# B&R Automation Studio project NAELD004C00R10L518F00 (part 24)

#### Act_Link.st
```iecst
(** 2019-01-07 **)
ACTION Act_Link:

	IF EDGEPOS(p_tyLinkUSSMEMA1AlmData.udiCode <> 0) THEN
		p_tyLinkUSSMEMA1AlmData.sProgNm	:= 'Mag1_1';
		p_tyLinkUSSMEMA1AlmData.sAlmMsg	:= 'Pulling Board Failed';
	END_IF

	IF EDGEPOS(p_tyLinkUSSMEMA2AlmData.udiCode <> 0) THEN
		p_tyLinkUSSMEMA2AlmData.sProgNm	:= 'Mag2_1';
		p_tyLinkUSSMEMA2AlmData.sAlmMsg	:= 'Pulling Board Failed';
	END_IF

	IF EDGEPOS(p_tyLinkUSSMEMA3AlmData.udiCode <> 0) THEN
		p_tyLinkUSSMEMA3AlmData.sProgNm	:= 'Mag3_1';
		p_tyLinkUSSMEMA3AlmData.sAlmMsg	:= 'Pulling Board Failed';
	END_IF

	IF EDGEPOS(p_tyLinkDSSMEMA1AlmData.udiCode <> 0) THEN
		p_tyLinkDSSMEMA1AlmData.sProgNm	:= 'Mag1_2';
		p_tyLinkDSSMEMA1AlmData.sAlmMsg	:= 'Pulling Board Failed';
	END_IF

	IF EDGEPOS(p_tyLinkDSSMEMA2AlmData.udiCode <> 0) THEN
		p_tyLinkDSSMEMA2AlmData.sProgNm	:= 'Mag2_2';
		p_tyLinkDSSMEMA2AlmData.sAlmMsg	:= 'Pulling Board Failed';
	END_IF

	IF EDGEPOS(p_tyLinkDSSMEMA3AlmData.udiCode <> 0) THEN
		p_tyLinkDSSMEMA3AlmData.sProgNm	:= 'Mag3_2';
		p_tyLinkDSSMEMA3AlmData.sAlmMsg	:= 'Pulling Board Failed';
	END_IF

	//Index 1 For Internal Use

	pa_tyAlmData[2]		:= p_tyLinkUsrFolderAlmData;
	pa_tyAlmData[3]		:= p_tyLinkLibVerAlmData;
	pa_tyAlmData[4]		:= p_tyLinkTimeAlmData;
	pa_tyAlmData[5]		:= p_tyLinkTimeAlmData1;
	pa_tyAlmData[6]		:= p_tyLinkHWInfoAlmData;
	pa_tyAlmData[7]		:= p_tyLinkProdRcpAlmData;
	pa_tyAlmData[8]		:= p_tyLinkMpProdRcpAlmData;
	pa_tyAlmData[9]		:= p_tyLinkMagRcpAlmData;
	pa_tyAlmData[10]	:= p_tyLinkMagRcpAlmData1;

	pa_tyAlmData[11]	:= p_tyLinkMcParamAlmData;
	pa_tyAlmData[12]	:= p_tyLinkNtParamAlmData;
	pa_tyAlmData[13]	:= p_tyLinkUsrMgmtAlmData;
	pa_tyAlmData[14]	:= p_tyLinkBuffer1AlmData;
	pa_tyAlmData[15]	:= p_tyLinkBuffer2AlmData;
	pa_tyAlmData[16]	:= p_tyLinkBuffer3AlmData;
	pa_tyAlmData[17]	:= p_tyLinkBuffer4AlmData;
	pa_tyAlmData[18]	:= p_tyLinkUSSMEMA1AlmData;
	pa_tyAlmData[19]	:= p_tyLinkUSSMEMA2AlmData;
	pa_tyAlmData[20]	:= p_tyLinkUSSMEMA3AlmData;
	pa_tyAlmData[21]	:= p_tyLinkUSSMEMA4AlmData;
	pa_tyAlmData[22]	:= p_tyLinkDSSMEMA1AlmData;
	pa_tyAlmData[23]	:= p_tyLinkDSSMEMA2AlmData;
	pa_tyAlmData[24]	:= p_tyLinkDSSMEMA3AlmData;
	pa_tyAlmData[25]	:= p_tyLinkDSSMEMA4AlmData;

	pa_tyAlmData[26]	:= p_tyLinkDSSMEMAAAlmData;
	pa_tyAlmData[27]	:= p_tyLinkDSSMEMABAlmData;
	pa_tyAlmData[28]	:= p_tyLinkInShutterAlmData;
	pa_tyAlmData[29]	:= p_tyLinkOutShutterAlmData;
	pa_tyAlmData[30]	:= p_tyLinkPullerAlmData;
	pa_tyAlmData[31]	:= p_tyLinkPullConvAlmData;
	pa_tyAlmData[32]	:= p_tyLinkMagConv1AlmData;
	pa_tyAlmData[33]	:= p_tyLinkMagConv2AlmData;
	pa_tyAlmData[34]	:= p_tyLinkMagConv3AlmData;
	pa_tyAlmData[35]	:= p_tyLinkMagConv4AlmData;

	pa_tyAlmData[36]	:= p_tyLinkAWOpenAlmData;
	pa_tyAlmData[37]	:= p_tyLinkAWOpenAlmData1;
	pa_tyAlmData[38]	:= p_tyLinkAWOpenAlmData2;
	pa_tyAlmData[39]	:= p_tyLinkAWOpenAlmData3;
	pa_tyAlmData[40]	:= p_tyLinkTravAlmData;
	pa_tyAlmData[41]	:= p_tyLinkTravAlmData1;
	pa_tyAlmData[42]	:= p_tyLinkTravAlmData2;
	pa_tyAlmData[43]	:= p_tyLinkTravAlmData3;
	pa_tyAlmData[44]	:= p_tyLinkLifterBtmAlmData;
	pa_tyAlmData[45]	:= p_tyLinkLifterBtmAlmData1;
	pa_tyAlmData[46]	:= p_tyLinkLifterBtmAlmData2;
	pa_tyAlmData[47]	:= p_tyLinkLifterBtmAlmData3;
	pa_tyAlmData[48]	:= p_tyLinkDIAlmData1;
	pa_tyAlmData[49]	:= p_tyLinkDIAlmData2;
	pa_tyAlmData[50]	:= p_tyLinkDIAlmData3;
	pa_tyAlmData[51]	:= p_tyLinkDIAlmData4;

	pa_tyAlmData[52]	:= p_tyLinkAGVMag1AlmData;
	pa_tyAlmData[53]	:= p_tyLinkAGVMag2AlmData;
	pa_tyAlmData[54]	:= p_tyLinkAGVMag3AlmData;
	pa_tyAlmData[55]	:= p_tyLinkAGVMag4AlmData;

	pa_tyAlmData[56]	:= p_tyLinkHermesAlmData;
	pa_tyAlmData[57]	:= p_tyLinkDSHermesAAlmData;
	pa_tyAlmData[58]	:= p_tyLinkDSHermesAAlmData1;
	pa_tyAlmData[59]	:= p_tyLinkDSHermesAAlmData2;
	pa_tyAlmData[60]	:= p_tyLinkDSHermesAAlmData3;
	pa_tyAlmData[61]	:= p_tyLinkDSHermesAAlmData4;

	pa_tyAlmData[62]	:= p_tyLinkDSHermesBAlmData;
	pa_tyAlmData[63]	:= p_tyLinkDSHermesBAlmData1;
	pa_tyAlmData[64]	:= p_tyLinkDSHermesBAlmData2;
	pa_tyAlmData[65]	:= p_tyLinkDSHermesBAlmData3;
	pa_tyAlmData[66]	:= p_tyLinkDSHermesBAlmData4;

	pa_tyAlmData[67]	:= p_tyLinkRmtHermesAlmData;
	pa_tyAlmData[68]	:= p_tyLinkRmtHermesAlmData1;
	pa_tyAlmData[69]	:= p_tyLinkRmtHermesAlmData2;
	pa_tyAlmData[70]	:= p_tyLinkRmtHermesAlmData3;
	pa_tyAlmData[71]	:= p_tyLinkLFLeaderAlmData;
	pa_tyAlmData[72]	:= p_tyLinkLFFollowerAlmData;
	pa_tyAlmData[73]	:= p_tyLinkLFFollowerInfoData;
	pa_tyAlmData[74]	:= p_tyLinkLFFollowerInfoData1;
	pa_tyAlmData[75]	:= p_tyLinkFollower1AlmData;
	pa_tyAlmData[76]	:= p_tyLinkFollower1InfoData;
	pa_tyAlmData[77]	:= p_tyLinkFollower1InfoData1;
	pa_tyAlmData[78]	:= p_tyLinkFollower2AlmData;
	pa_tyAlmData[79]	:= p_tyLinkFollower2InfoData;
	pa_tyAlmData[80]	:= p_tyLinkFollower2InfoData1;
	pa_tyAlmData[81]	:= p_tyLinkLCSMngRcpAlmData;
	pa_tyAlmData[82]	:= p_tyLinkLCSLFAlmData;
	pa_tyAlmData[83]	:= p_tyLinkLCSLFInfoData;
	pa_tyAlmData[84]	:= p_tyLinkOpsTravLifLDAlmData;

	pa_tyAlmData[85]	:= p_tyLinkPPAlmData;
	pa_tyAlmData[86]	:= p_tyLinkPPAlmData1;
	pa_tyAlmData[87]	:= p_tyLinkPPAlmData2;
	pa_tyAlmData[89]	:= p_tyLinkPPAlmData3;
//	pa_tyAlmData[90]	:= p_tyLinkOpsMagLD3AlmData;
//	pa_tyAlmData[91]	:= p_tyLinkOpsMagLD3AlmData1;
//	pa_tyAlmData[92]	:= p_tyLinkOpsMagLD4AlmData;
//	pa_tyAlmData[93]	:= p_tyLinkOpsMagLD4AlmData1;
	pa_tyAlmData[94]	:= p_tyLinkOpsLifMagLDAlmData;
	pa_tyAlmData[95]	:= p_tyLinkOpsLifMagLDAlmData1;

	pa_tyAlmData[96]	:= p_tyLinkOpsMagConvLD1AlmData;
	pa_tyAlmData[97]	:= p_tyLinkOpsMagConvLD1AlmData1;
	pa_tyAlmData[98]	:= p_tyLinkOpsMagConvLD2AlmData;
	pa_tyAlmData[99]	:= p_tyLinkOpsMagConvLD2AlmData1;
	pa_tyAlmData[100]	:= p_tyLinkOpsMagConvLD3AlmData;
	pa_tyAlmData[101]	:= p_tyLinkOpsMagConvLD3AlmData1;
	pa_tyAlmData[102]	:= p_tyLinkOpsMagConvLD4AlmData;
	pa_tyAlmData[103]	:= p_tyLinkOpsMagConvLD4AlmData1;

	pa_tyAlmData[104]	:= p_tyLinkSelClamp1AlmData;
	pa_tyAlmData[105]	:= p_tyLinkSelClamp2AlmData;
	pa_tyAlmData[106]	:= p_tyLinkSelClamp3AlmData;
	pa_tyAlmData[107]	:= p_tyLinkSelClamp4AlmData;

	pa_tyAlmData[108]	:= p_tyLinkUSSOT1AlmData;
	pa_tyAlmData[109]	:= p_tyLinkUSSOT2AlmData;
	pa_tyAlmData[110]	:= p_tyLinkUSSOT3AlmData;
	pa_tyAlmData[111]	:= p_tyLinkUSSOT4AlmData;
	pa_tyAlmData[112]	:= p_tyLinkDSSOT1AlmData;
	pa_tyAlmData[113]	:= p_tyLinkDSSOT2AlmData;
	pa_tyAlmData[114]	:= p_tyLinkDSSOT3AlmData;
	pa_tyAlmData[115]	:= p_tyLinkDSSOT4AlmData;

	pa_tyAlmData[116]	:= p_tyLinkMcAlarmData;
	pa_tyAlmData[117]	:= p_tyLinkMc1AlarmData;

	pa_tyAlmData[118]	:= p_tyLinkUSBBarcodeAlmData;
	pa_tyAlmData[119]	:= p_tyLinkUSBBarcodeAlmData1;
	pa_tyAlmData[120]	:= p_tyLinkUSBBarcodeAlmData2;

	pa_tyAlmData[121]	:= p_tyLinkAGVAlmData1;
	pa_tyAlmData[122]	:= p_tyLinkRS232FrmAlmData;

	pa_tyAlmData[123]	:= p_tyLinkAWPushOrPullerAlmData;
	pa_tyAlmData[124]	:= p_tyLinkAWPushOrPullerAlmData1;
	pa_tyAlmData[125]	:= p_tyLinkAWPushOrPullerAlmData2;
	pa_tyAlmData[126]	:= p_tyLinkAWPushOrPullerAlmData3;
	pa_tyAlmData[127]	:= p_tyLinkMtrPshrAlmData;

	pa_tyAlmData[128]	:= p_tyLinkInShutterAlmData2;
	pa_tyAlmData[129]	:= p_tyLinkInShutterAlmData3;

	pa_tyAlmData[130]	:= p_tyLinkDIAlmData5;
	pa_tyAlmData[131]	:= p_tyLinkDIAlmData6;		//JOHN

//	pa_tyAlmData[131]	:= p_tyLinkUSHermesInfoData1;//new for Hermes 1.3
//	pa_tyAlmData[132]	:= p_tyLinkUSHermesInfoData2;//new for Hermes 1.3
//	pa_tyAlmData[133]	:= p_tyLinkUSHermesAlmData5;//new for Hermes 1.3
	pa_tyAlmData[134]	:= p_tyLinkRmtHermesInfoData;//new for Hermes 1.3
	pa_tyAlmData[135]	:= p_tyLinkSvyHermesAlmData;//new for Hermes 1.3
	pa_tyAlmData[136]	:= p_tyLinkSvyHermesAlmData1;//new for Hermes 1.3
	pa_tyAlmData[137]	:= p_tyLinkSvyHermesAlmData2;//new for Hermes 1.3
	pa_tyAlmData[138]	:= p_tyLinkSvyHermesAlmData3;//new for Hermes 1.3
	pa_tyAlmData[139]	:= p_tyLinkSvyHermesInfoData;//new for Hermes 1.3
	pa_tyAlmData[140]	:= p_tyLinkSvyHermesInfoData1;//new for Hermes 1.3
	pa_tyAlmData[141]	:= p_tyLinkSvyHermesInfoData2;//new for Hermes 1.3
	pa_tyAlmData[142]	:= p_tyLinkSvyHermesInfoData3;//new for Hermes 1.3
	pa_tyAlmData[143]	:= p_tyLinkSvyHermesAlmData4;//new for Hermes 1.3
	pa_tyAlmData[144]	:= p_tyLinkSvyHermesInfoData4;//new for Hermes 1.3

	pa_tyAlmData[145]	:= p_tyLinkAutoRcpAlmData;
	pa_tyAlmData[146]	:= p_tyLinkAutoRcpInfoData;
	pa_tyAlmData[147]	:= p_tyLinkAutoRcpInfoData1;
	pa_tyAlmData[148]	:= p_tyLinkOutShutterAlmData2;
	pa_tyAlmData[149]	:= p_tyLinkTrllyAlmData;
	pa_tyAlmData[150]	:= p_tyLinkTrlly2AlmData;

END_ACTION
```

#### Act_LinkAction.st
```iecst
(** 2019-03-29 **)
ACTION Act_LinkAction:

	//Delete Old Log File for 24 hours After Machine is Continuous Running 30 Days.

	fbDlyTmr(IN := TRUE);
	IF fbDlyTmr.Q THEN
		fbDeleteLogTmr (IN := TRUE);
		IF fbDeleteLogTmr.Q AND eStatus <> Busy THEN
			p_eAct := AlarmActDeleteOldLog;
			IF eStat = AlarmActDeleteOldLog AND eStatus = Done THEN
				p_eAct := AlarmActIdle;
				fbDlyTmr (IN := FALSE);
				fbDeleteLogTmr (IN := FALSE);
			END_IF
		END_IF
	END_IF

END_ACTION
```

#### Act_Main.st
```iecst
(** 2019-02-23 **)
ACTION Act_Main:

	//Main
	CASE eStat OF

		AlarmActIdle:
			IF eStatus <> Idle THEN	//Reset Data
				//Private
				fbDirCreate1(bEn := FALSE);
				fbDirCreate2(bEn := FALSE);
				fbFileOldDel1(bEn := FALSE);
				fbFileRead1(bEn := FALSE);
				fbFileAppend1(bEn := FALSE);
				fbFileWrite1(bEn := FALSE);
				usiStep	:= 0;

				bHistoryFileNotFound	:= FALSE;
				udiWriteLogCntr			:= 1;

				sStatTxt	:= a_sStatText[eStat];

			END_IF

			eStatus	:= Idle;

		AlarmActCreateDir:
			IF eStatus = Idle OR eStatus = Busy THEN

				eStatus	:= Busy;

				sStatTxt	:= a_sStatText[eStat];

				CASE usiStep OF
					0:
						fbDirCreate1(bEn := TRUE);
						IF fbDirCreate1.udiStatus = 0 THEN
							usiStep	:= 1;
						ELSIF fbDirCreate1.udiStatus < 65534 THEN
							eStatus		:= Error;

							IF fbDirCreate1.udiStatus = 1908 THEN
								udiStatus	:= 10000;	//Create User Directory Error
							ELSE
								udiStatus	:= fbDirCreate1.udiStatus;
							END_IF
						END_IF

					1:
						fbDirCreate2(bEn := TRUE);
						IF fbDirCreate2.udiStatus = 0 THEN
							eStatus	:= Done;
						ELSIF fbDirCreate2.udiStatus < 65534 THEN
							eStatus		:= Error;

							IF fbDirCreate2.udiStatus = 1908 THEN
								udiStatus	:= 10001;	//Create Alarm Directory Error
							ELSE
								udiStatus	:= fbDirCreate2.udiStatus;
							END_IF
						END_IF

				END_CASE

			END_IF

		AlarmActDeleteOldLog:
			IF eStatus = Idle OR eStatus = Busy THEN

				eStatus	:= Busy;

				sStatTxt	:= a_sStatText[eStat];

				fbFileOldDel1.dtDTNow			:= p_dtCurrDT;
				fbFileOldDel1.udiFileKeepDay	:= p_udiFileKeepDay;
				fbFileOldDel1(bEn := TRUE);
				IF fbFileOldDel1.udiStatus = 0 THEN
					eStatus	:= Done;
				ELSIF fbFileOldDel1.udiStatus < 65534 THEN
					eStatus		:= Error;

					IF fbFileOldDel1.udiStatus = 1910 THEN
						udiStatus	:= 10002;	//Get Directory Info Error While Deleting Old Log
					ELSIF fbFileOldDel1.udiStatus = 1911 THEN
						udiStatus	:= 10003;	//Directory Read Error While Deleting Old Log
					ELSIF fbFileOldDel1.udiStatus = 1912 THEN
						udiStatus	:= 10004;	//File Delete Error While Deleting Old Log
					ELSE
						udiStatus	:= fbFileOldDel1.udiStatus;
					END_IF
				END_IF

			END_IF

		AlarmActReadHistory:
			IF eStatus = Idle OR eStatus = Busy THEN

				eStatus	:= Busy;

				sStatTxt	:= a_sStatText[eStat];

				fbFileRead1(bEn := TRUE);
				IF fbFileRead1.udiStatus = 0 THEN
					eStatus	:= Done;
				ELSIF fbFileRead1.udiStatus < 65534 THEN
					eStatus		:= Error;

					IF fbFileRead1.udiStatus = 1900 THEN
						udiStatus	:= 10005;	//File Open Error While Reading Alarm History
					ELSIF fbFileRead1.udiStatus = 1902 THEN
						udiStatus	:= 10006;	//File Read Error While Reading Alarm History
					ELSIF fbFileRead1.udiStatus = 1904 THEN
						udiStatus	:= 10007;	//File Close Error While Reading Alarm History
					ELSIF fbFileRead1.udiStatus = 1915 THEN
						eStatus					:= Done;
						bHistoryFileNotFound	:= TRUE;
					ELSE
						udiStatus	:= fbFileRead1.udiStatus;
					END_IF
				END_IF

			END_IF

		AlarmActWriteHistory:
			IF eStatus = Idle OR eStatus = Busy THEN

				eStatus	:= Busy;

				sStatTxt	:= a_sStatText[eStat];

				fbFileWrite1(bEn := TRUE);
				IF fbFileWrite1.udiStatus = 0 THEN
					eStatus	:= Done;
				ELSIF fbFileWrite1.udiStatus < 65534 THEN
					eStatus		:= Error;

					IF fbFileWrite1.udiStatus = 1900 THEN
						udiStatus	:= 10008;	//File Open Error While Writing Alarm History
					ELSIF fbFileWrite1.udiStatus = 1901 THEN
						udiStatus	:= 10009;	//File Create Error While Writing Alarm History
					ELSIF fbFileWrite1.udiStatus = 1903 THEN
						udiStatus	:= 10010;	//File Write Error While Writing Alarm History
					ELSIF fbFileWrite1.udiStatus = 1904 THEN
						udiStatus	:= 10011;	//File Close Error While Writing Alarm History
					ELSIF fbFileWrite1.udiStatus = 1914 THEN
						udiStatus	:= 10012;	//Directory Does Not Exist While Writing Alarm History
					ELSE
						udiStatus	:= fbFileWrite1.udiStatus;
					END_IF
				END_IF

			END_IF

		AlarmActAppendLog:
			IF eStatus = Idle OR eStatus = Busy THEN

				eStatus	:= Busy;

				sStatTxt	:= a_sStatText[eStat];

				dtCurrDTTemp			:= p_dtCurrDT;
				fbFileAppend1.sFile		:= DT_TO_STRING(dtCurrDTTemp);
				fbFileAppend1.sFile		:= MID(fbFileAppend1.sFile , 10 , 4);
				fbFileAppend1.sFile		:= CONCAT('ALARM_' , fbFileAppend1.sFile);
				fbFileAppend1.sFile		:= CONCAT(fbFileAppend1.sFile , '.dat');

				fbFileAppend1.p_Src		:= ADR(a_sLogList[udiWriteLogCntr]);
				fbFileAppend1.udiLen	:= LEN(a_sLogList[udiWriteLogCntr]);

				fbFileAppend1(bEn := TRUE);
				IF fbFileAppend1.udiStatus = 0 THEN
					IF udiWriteLogCntr >= udiLogCntr THEN
						eStatus	:= Done;
					ELSE
						udiWriteLogCntr	:= udiWriteLogCntr + 1;
						fbFileAppend1(bEn := FALSE);
					END_IF

				ELSIF fbFileAppend1.udiStatus < 65534 THEN
					eStatus		:= Error;

					IF fbFileAppend1.udiStatus = 1900 THEN
						udiStatus	:= 10013;	//File Open Error While Writing Alarm Log
					ELSIF fbFileAppend1.udiStatus = 1901 THEN
						udiStatus	:= 10014;	//File Create Error While Writing Alarm Log
					ELSIF fbFileAppend1.udiStatus = 1913 THEN
						udiStatus	:= 10015;	//Get File Info Error While Writing Alarm Log
					ELSIF fbFileAppend1.udiStatus = 1903 THEN
						udiStatus	:= 10016;	//File Write Error While Writing Alarm Log
					ELSIF fbFileAppend1.udiStatus = 1904 THEN
						udiStatus	:= 10017;	//File Close Error While Writing Alarm Log
					ELSIF fbFileAppend1.udiStatus = 1914 THEN
						udiStatus	:= 10018;	//Directory Does Not Exist While Writing Alarm Log
					ELSE
						udiStatus	:= fbFileAppend1.udiStatus;
					END_IF
				END_IF

			END_IF

		AlarmActAppendLogWriteHistory:
			IF eStatus = Idle OR eStatus = Busy THEN

				eStatus	:= Busy;

				sStatTxt	:= a_sStatText[eStat];

				dtCurrDTTemp			:= p_dtCurrDT;
				fbFileAppend1.sFile		:= DT_TO_STRING(dtCurrDTTemp);
				fbFileAppend1.sFile		:= MID(fbFileAppend1.sFile , 10 , 4);
				fbFileAppend1.sFile		:= CONCAT('ALARM_' , fbFileAppend1.sFile);
				fbFileAppend1.sFile		:= CONCAT(fbFileAppend1.sFile , '.dat');

				fbFileAppend1.p_Src		:= ADR(a_sLogList[udiWriteLogCntr]);
				fbFileAppend1.udiLen	:= LEN(a_sLogList[udiWriteLogCntr]);

				fbFileAppend1(bEn := TRUE);
				fbFileWrite1(bEn := TRUE);

				IF (fbFileAppend1.udiStatus = 0) AND (udiWriteLogCntr >= udiLogCntr) AND fbFileWrite1.udiStatus = 0 THEN
					eStatus	:= Done;

				ELSIF fbFileAppend1.udiStatus = 0 AND udiWriteLogCntr < udiLogCntr THEN
					udiWriteLogCntr	:= udiWriteLogCntr + 1;
					fbFileAppend1(bEn := FALSE);

				ELSIF fbFileWrite1.udiStatus > 0 AND fbFileWrite1.udiStatus < 65534 THEN
					eStatus		:= Error;

					IF fbFileWrite1.udiStatus = 1900 THEN
						udiStatus	:= 10019;	//File Open Error While Writing Alarm History
					ELSIF fbFileWrite1.udiStatus = 1901 THEN
						udiStatus	:= 10020;	//File Create Error While Writing Alarm History
					ELSIF fbFileWrite1.udiStatus = 1903 THEN
						udiStatus	:= 10021;	//File Write Error While Writing Alarm History
					ELSIF fbFileWrite1.udiStatus = 1904 THEN
						udiStatus	:= 10022;	//File Close Error While Writing Alarm History
					ELSIF fbFileWrite1.udiStatus = 1914 THEN
						udiStatus	:= 10023;	//Directory Does Not Exist While Writing Alarm History
					ELSE
						udiStatus	:= fbFileWrite1.udiStatus;
					END_IF

				ELSIF fbFileAppend1.udiStatus > 0 AND fbFileAppend1.udiStatus < 65534 THEN
					eStatus		:= Error;

					IF fbFileAppend1.udiStatus = 1900 THEN
						udiStatus	:= 10024;	//File Open Error While Writing Alarm Log
					ELSIF fbFileAppend1.udiStatus = 1901 THEN
						udiStatus	:= 10025;	//File Create Error While Writing Alarm Log
					ELSIF fbFileAppend1.udiStatus = 1913 THEN
						udiStatus	:= 10026;	//Get File Info Error While Writing Alarm Log
					ELSIF fbFileAppend1.udiStatus = 1903 THEN
						udiStatus	:= 10027;	//File Write Error While Writing Alarm Log
					ELSIF fbFileAppend1.udiStatus = 1904 THEN
						udiStatus	:= 10028;	//File Close Error While Writing Alarm Log
					ELSIF fbFileAppend1.udiStatus = 1914 THEN
						udiStatus	:= 10029;	//Directory Does Not Exist While Writing Alarm Log
					ELSE
						udiStatus	:= fbFileAppend1.udiStatus;
					END_IF
				END_IF

			END_IF

		AlarmActResetHistory:
			IF eStatus = Idle OR eStatus = Busy THEN

				eStatus	:= Busy;

				sStatTxt	:= a_sStatText[eStat];

				memset(ADR(a_sHistoryList) , 0 , SIZEOF(a_sHistoryList));

				fbFileWrite1(bEn := TRUE);
				IF fbFileWrite1.udiStatus = 0 THEN
					eStatus	:= Done;
				ELSIF fbFileWrite1.udiStatus < 65534 THEN
					eStatus		:= Error;

					IF fbFileWrite1.udiStatus = 1900 THEN
						udiStatus	:= 10030;	//File Open Error While Resetting Alarm History
					ELSIF fbFileWrite1.udiStatus = 1901 THEN
						udiStatus	:= 10031;	//File Create Error While Resetting Alarm History
					ELSIF fbFileWrite1.udiStatus = 1903 THEN
						udiStatus	:= 10032;	//File Write Error While Resetting Alarm History
					ELSIF fbFileWrite1.udiStatus = 1904 THEN
						udiStatus	:= 10033;	//File Close Error While Resetting Alarm History
					ELSIF fbFileWrite1.udiStatus = 1914 THEN
						udiStatus	:= 10034;	//Directory Does Not Exist While Resetting Alarm History
					ELSE
						udiStatus	:= fbFileWrite1.udiStatus;
					END_IF
				END_IF

			END_IF

		AlarmActBGStartLog:
			IF eStatus = Idle OR eStatus = Busy THEN

				sStatTxt	:= a_sStatText[eStat];

				bAlarmLog	:= TRUE;
				eStatus		:= Done;

			END_IF

		AlarmActBGStopLog:
			IF eStatus = Idle OR eStatus = Busy THEN

				sStatTxt	:= a_sStatText[eStat];

				bAlarmLog	:= FALSE;
				eStatus		:= Done;

			END_IF

	END_CASE

END_ACTION
```

#### Act_RstErr.st
```iecst
(** 2020-07-27 **)
ACTION Act_RstErr:

	IF p_udiRstErr <> udiRstErrOld THEN
		bRstErr			:= TRUE;
		udiRstErrOld	:= p_udiRstErr;
	ELSE
		bRstErr			:= FALSE;
	END_IF

	//Checking which Warning is clear
	IF a_tyWarningCurrList[1].sMsg <> '' AND p_tyLinkLibVerAlmData.udiCode = 0 THEN

		FOR udi2 := 1 TO (udiWarningMax) DO
			udiRecorded1:= udiRecorded[udi2];
			IF 	(pa_tyAlmData[udiRecorded1].eSeverity =  AlmSeverityNA) AND udiRecorded1<> 0 THEN
				bRstWarning := TRUE;
				EXIT;
			ELSE
				bRstWarning := FALSE;
			END_IF

		END_FOR
	ELSE
		bRstWarning := FALSE;
	END_IF

END_ACTION
```

### ProdRcp.typ
```iecst
(*2020-07-24*)
(**)
(*Action*)

TYPE
	eProdRcpAction :
		(
		ProdRcpActIdle,
		ProdRcpActCreateDir,
		ProdRcpActAddEdit,
		ProdRcpActDel,
		ProdRcpActGetInfo,
		ProdRcpActGetList,
		ProdRcpActFilter,
		ProdRcpActLoadRcp,
		ProdRcpActAdd,
		ProdRcpActEdit,
		ProdRcpActReadCurrRcp,
		ProdRcpActWriteCurrRcpParam,
		ProdRcpActSaveList,
		ProdRcpActSort,
		ProdRcpActEndCharFilter
		);
END_TYPE

(**)
(*Data*)

TYPE
	tyProdRcpParam : 	STRUCT
		sRcpNm : STRING[254];
		diWidthInUM : DINT;
		diWidthInUM2 : DINT;
		diIntvlCntr : DINT;
		diMinSltValue : DINT;
		diMaxSltValue : DINT;
		diPitch : DINT;
		usiMcMod : USINT;
		usiFlippedBrd : USINT;
		bTopToBtm : BOOL;
		bLongBrd : BOOL;
		sDisplayInfo : STRING[30];
		dtLastModified : DATE_AND_TIME;
		diWidthInUMRear : DINT;
		diPitchRear : DINT;
		diMinSltValueRear : DINT;
		diMaxSltValueRear : DINT;
		diMtrPshrExtSpd : DINT; (*Puller*)
		diMtrPshrExtTorq : DINT;
		diPshrOffset : DINT;
	END_STRUCT;
END_TYPE
```

### ProdRcp.var
```iecst
(*2020-06-08*)
(**)
(*Constant*)
VAR CONSTANT
	c_udiProdRcpMax : UDINT := 2000;
END_VAR
(**)
(*Action & State & Status*)
VAR
	p_ProdRcpStat : UDINT;
	p_ProdRcpStatus : UDINT;
	p_ProdRcpStatTxt : UDINT;
END_VAR
(**)
(*Alarm*)
VAR
	p_ProdRcpAlmData : UDINT;
END_VAR
(**)
(*Output*)
VAR
	p_ProdRcpNmExist : UDINT;
	p_ProdRcpNmNotExist : UDINT;
	p_ProdRcpNmEmpty : UDINT;
	p_ProdRcpListFull : UDINT;
	p_ProdRcpCurrList : UDINT;
	p_ProdRcpFilterList : UDINT;
	p_ProdRcpSortedList : UDINT;
	p_ProdRcpScanList : UDINT;
	p_ProdRcpInfoOut : UDINT;
	p_ProdRcpFileNotFound : UDINT;
	p_ProdRcpCurrRcpAll : UDINT;
END_VAR
(**)
VAR
	p_ProdRcpCurrRcp0 : UDINT;
	p_ProdRcpCurrRcp0Nm : UDINT;
	p_ProdRcpCurrRcp0Width : UDINT;
	p_ProdRcpCurrRcp0MinSltValue : UDINT;
	p_ProdRcpCurrRcp0MaxSltValue : UDINT;
	p_ProdRcpCurrRcp0Pitch : UDINT;
	p_ProdRcpCurrRcp0McMod : UDINT;
	p_ProdRcpCurrRcp0FlippedBrd : UDINT;
	p_ProdRcpCurrRcp0TopToBtm : UDINT;
	p_ProdRcpCurrRcp0LongBrd : UDINT;
	p_ProdRcpCurrRcp0DisplayInfo : UDINT;
	p_ProdRcpCurrRcp0LastModified : UDINT;
	p_ProdRcpCurrRcp0Width2 : UDINT;
	p_ProdRcpCurrRcp0WidthRear : UDINT;
	p_ProdRcpCurrRcp0PitchRear : UDINT;
	p_ProdRcpCurrRcp0MinSltRear : UDINT;
	p_ProdRcpCurrRcp0MaxSltRear : UDINT;
	p_ProdRcpCurrRcp0PshrOffset : UDINT;
	p_ProdRcpCurrRcp0MtrPshrExtSpd : UDINT;
	p_ProdRcpCurrRcp0MtrPshrExtTorq : UDINT;
END_VAR
(**)
VAR
	p_ProdRcpCurrRcp1 : UDINT;
	p_ProdRcpCurrRcp1Nm : UDINT;
	p_ProdRcpCurrRcp1Width : UDINT;
	p_ProdRcpCurrRcp1MinSltValue : UDINT;
	p_ProdRcpCurrRcp1MaxSltValue : UDINT;
	p_ProdRcpCurrRcp1Pitch : UDINT;
	p_ProdRcpCurrRcp1McMod : UDINT;
	p_ProdRcpCurrRcp1FlippedBrd : UDINT;
	p_ProdRcpCurrRcp1TopToBtm : UDINT;
	p_ProdRcpCurrRcp1LongBrd : UDINT;
	p_ProdRcpCurrRcp1DisplayInfo : UDINT;
	p_ProdRcpCurrRcp1LastModified : UDINT;
	p_ProdRcpCurrRcp1Width2 : UDINT;
	p_ProdRcpCurrRcp1WidthRear : UDINT;
	p_ProdRcpCurrRcp1PitchRear : UDINT;
	p_ProdRcpCurrRcp1MinSltRear : UDINT;
	p_ProdRcpCurrRcp1MaxSltRear : UDINT;
	p_ProdRcpCurrRcp1PshrOffset : UDINT;
	p_ProdRcpCurrRcp1MtrPshrExtSpd : UDINT;
	p_ProdRcpCurrRcp1MtrPshrExtTorq : UDINT;
END_VAR
(**)
VAR
	p_ProdRcpCurrRcp2 : UDINT;
	p_ProdRcpCurrRcp2Nm : UDINT;
	p_ProdRcpCurrRcp2Width : UDINT;
	p_ProdRcpCurrRcp2MinSltValue : UDINT;
	p_ProdRcpCurrRcp2MaxSltValue : UDINT;
	p_ProdRcpCurrRcp2Pitch : UDINT;
	p_ProdRcpCurrRcp2McMod : UDINT;
	p_ProdRcpCurrRcp2FlippedBrd : UDINT;
	p_ProdRcpCurrRcp2TopToBtm : UDINT;
	p_ProdRcpCurrRcp2LongBrd : UDINT;
	p_ProdRcpCurrRcp2DisplayInfo : UDINT;
	p_ProdRcpCurrRcp2LastModified : UDINT;
	p_ProdRcpCurrRcp2Width2 : UDINT;
	p_ProdRcpCurrRcp2WidthRear : UDINT;
	p_ProdRcpCurrRcp2PitchRear : UDINT;
	p_ProdRcpCurrRcp2MinSltRear : UDINT;
	p_ProdRcpCurrRcp2MaxSltRear : UDINT;
	p_ProdRcpCurrRcp2PshrOffset : UDINT;
	p_ProdRcpCurrRcp2MtrPshrExtSpd : UDINT;
	p_ProdRcpCurrRcp2MtrPshrExtTorq : UDINT;
END_VAR
(**)
VAR
	p_ProdRcpCurrRcp3 : UDINT;
	p_ProdRcpCurrRcp3Nm : UDINT;
	p_ProdRcpCurrRcp3Width : UDINT;
	p_ProdRcpCurrRcp3MinSltValue : UDINT;
	p_ProdRcpCurrRcp3MaxSltValue : UDINT;
	p_ProdRcpCurrRcp3Pitch : UDINT;
	p_ProdRcpCurrRcp3McMod : UDINT;
	p_ProdRcpCurrRcp3FlippedBrd : UDINT;
	p_ProdRcpCurrRcp3TopToBtm : UDINT;
	p_ProdRcpCurrRcp3LongBrd : UDINT;
	p_ProdRcpCurrRcp3DisplayInfo : UDINT;
	p_ProdRcpCurrRcp3LastModified : UDINT;
	p_ProdRcpCurrRcp3Width2 : UDINT;
	p_ProdRcpCurrRcp3WidthRear : UDINT;
	p_ProdRcpCurrRcp3PitchRear : UDINT;
	p_ProdRcpCurrRcp3MinSltRear : UDINT;
	p_ProdRcpCurrRcp3MaxSltRear : UDINT;
	p_ProdRcpCurrRcp3PshrOffset : UDINT;
	p_ProdRcpCurrRcp3MtrPshrExtSpd : UDINT;
	p_ProdRcpCurrRcp3MtrPshrExtTorq : UDINT;
END_VAR
(**)
VAR
	p_ProdRcpCurrRcp4 : UDINT;
	p_ProdRcpCurrRcp4Nm : UDINT;
	p_ProdRcpCurrRcp4Width : UDINT;
	p_ProdRcpCurrRcp4MinSltValue : UDINT;
	p_ProdRcpCurrRcp4MaxSltValue : UDINT;
	p_ProdRcpCurrRcp4Pitch : UDINT;
	p_ProdRcpCurrRcp4McMod : UDINT;
	p_ProdRcpCurrRcp4FlippedBrd : UDINT;
	p_ProdRcpCurrRcp4TopToBtm : UDINT;
	p_ProdRcpCurrRcp4LongBrd : UDINT;
	p_ProdRcpCurrRcp4DisplayInfo : UDINT;
	p_ProdRcpCurrRcp4LastModified : UDINT;
	p_ProdRcpCurrRcp4Width2 : UDINT;
	p_ProdRcpCurrRcp4WidthRear : UDINT;
	p_ProdRcpCurrRcp4PitchRear : UDINT;
	p_ProdRcpCurrRcp4MinSltRear : UDINT;
	p_ProdRcpCurrRcp4MaxSltRear : UDINT;
	p_ProdRcpCurrRcp4PshrOffset : UDINT;
	p_ProdRcpCurrRcp4MtrPshrExtSpd : UDINT;
	p_ProdRcpCurrRcp4MtrPshrExtTorq : UDINT;
END_VAR
(**)
VAR
	p_ProdRcpCurrRcp5 : UDINT;
	p_ProdRcpCurrRcp5Nm : UDINT;
	p_ProdRcpCurrRcp5Width : UDINT;
	p_ProdRcpCurrRcp5MinSltValue : UDINT;
	p_ProdRcpCurrRcp5MaxSltValue : UDINT;
	p_ProdRcpCurrRcp5Pitch : UDINT;
	p_ProdRcpCurrRcp5McMod : UDINT;
	p_ProdRcpCurrRcp5FlippedBrd : UDINT;
	p_ProdRcpCurrRcp5TopToBtm : UDINT;
	p_ProdRcpCurrRcp5LongBrd : UDINT;
	p_ProdRcpCurrRcp5DisplayInfo : UDINT;
	p_ProdRcpCurrRcp5LastModified : UDINT;
	p_ProdRcpCurrRcp5Width2 : UDINT;
	p_ProdRcpCurrRcp5WidthRear : UDINT;
	p_ProdRcpCurrRcp5PitchRear : UDINT;
	p_ProdRcpCurrRcp5MinSltRear : UDINT;
	p_ProdRcpCurrRcp5MaxSltRear : UDINT;
	p_ProdRcpCurrRcp5PshrOffset : UDINT;
	p_ProdRcpCurrRcp5MtrPshrExtSpd : UDINT;
	p_ProdRcpCurrRcp5MtrPshrExtTorq : UDINT;
END_VAR
```

### Program Logical/ProdRcp/ProdRcp

#### InputRef_Link.var
```iecst
(*2019-04-24*)
(**)
VAR
	rWidthInMM : REAL;
	rWidthInMM2 : REAL;
	sWidthInMM : STRING[30];
	sWidthInMM2 : STRING[30];
	sWidthInMMRear : STRING[30];
	p_bLinkStartupRun : REFERENCE TO BOOL;
	p_bLinkNtParamLCSManageRcpPrep : REFERENCE TO BOOL;
	p_bLinkMcParamLCSManageRcpEn : REFERENCE TO BOOL;
	p_eLinkLCSMngRcpProdRcpAct : REFERENCE TO eProdRcpAction;
	p_eLinkUIProdRcpAct : REFERENCE TO eProdRcpAction;
	p_eLinkMag : REFERENCE TO eLDMag;
	rWidthInMMRear : REAL;
END_VAR
```

#### Local.var
```iecst
(*2020-07-24*)
(**)
(*Local Action, State & Status*)
VAR
	eAct : eProdRcpAction := ProdRcpActIdle;
	eStat : eProdRcpAction := ProdRcpActIdle;
	eStatus : eFBStatus := Idle;
	udiStatus : UDINT := 0;
	sStatTxt : STRING[200] := '';
	a_sStatText : ARRAY[0..50] OF STRING[200] := ['Idling','Creating Directory','Adding and Editing Files','Deleting Files','Get Info','Get List','Filtering Files','Loading Recipe','Adding Files','Editing Files','Reading Current Recipe','Writing Current Recipe Parameter','Saving Recipe List',38('')];
END_VAR
(**)
(*Local Alarm*)
VAR
	tyAlmData : tyAlmDat;
	a_tyAlmText : ARRAY[10000..10099] OF tyAlmTxt := [(sAlmText:='Create User Directory Error',sRcyText:='Unable To Create User Directory. Please Contact Nutek For A Possible Solution'),(sAlmText:='Create Product Recipe Directory Error',sRcyText:='Unable To Create Product Recipe Directory. Please Contact Nutek For A Possible Solution'),(sAlmText:='File Open Error While Adding & Editing',sRcyText:='An Error Was Encountered While Trying To Open File. Please Contact Nutek For A Possible Solution.'),(sAlmText:='File Create Error While Adding & Editing',sRcyText:='An Error Was Encountered While Trying To Create File. Please Contact Nutek For A Possible Solution.'),(sAlmText:='File Write Error While Adding & Editing',sRcyText:='An Error Was Encountered While Trying To Write File. Please Contact Nutek For A Possible Solution.'),(sAlmText:='File Close Error While Adding & Editing',sRcyText:='An Error Was Encountered While Trying To Close File. Please Contact Nutek For A Possible Solution.'),(sAlmText:='File Open Error While Deleting',sRcyText:='An Error Was Encountered While Trying To Open File. Please Contact Nutek For A Possible Solution.'),(sAlmText:='File Create Error While Deleting',sRcyText:='An Error Was Encountered While Trying To Create File. Please Contact Nutek For A Possible Solution.'),(sAlmText:='File Write Error While Deleting',sRcyText:='An Error Was Encountered While Trying To Write File. Please Contact Nutek For A Possible Solution.'),(sAlmText:='File Close Error While Deleting',sRcyText:='An Error Was Encountered While Trying To Close File. Please Contact Nutek For A Possible Solution.'),(sAlmText:='File Open Error While Getting List',sRcyText:='An Error Was Encountered While Trying To Open File. Please Contact Nutek For A Possible Solution.'),(sAlmText:='File Read Error While Getting List',sRcyText:='An Error Was Encountered While Trying To Read File. Please Contact Nutek For A Possible Solution.'),(sAlmText:='File Close Error While Getting List',sRcyText:='An Error Was Encountered While Trying To Close File. Please Contact Nutek For A Possible Solution.'),(sAlmText:='Directory Does Not Exist While Adding & Editing',sRcyText:='The Directory Does Not Exist.Please Contact Nutek For A Possible Solution.'),(sAlmText:='Directory Does Not Exist While Deleting',sRcyText:='The Directory Does Not Exist.Please Contact Nutek For A Possible Solution.'),(sAlmText:='File Open Error While Adding',sRcyText:='An Error Was Encountered While Trying To Open File. Please Contact Nutek For A Possible Solution.'),(sAlmText:='File Create Error While Adding',sRcyText:='An Error Was Encountered While Trying To Create File. Please Contact Nutek For A Possible Solution.'),(sAlmText:='File Write Error While Adding',sRcyText:='An Error Was Encountered While Trying To Write File. Please Contact Nutek For A Possible Solution.'),(sAlmText:='File Close Error While Adding',sRcyText:='An Error Was Encountered While Trying To Close File. Please Contact Nutek For A Possible Solution.'),(sAlmText:='Directory Does Not Exist While Adding',sRcyText:='The Directory Does Not Exist.Please Contact Nutek For A Possible Solution.'),(sAlmText:='File Open Error While Editing',sRcyText:='An Error Was Encountered While Trying To Open File. Please Contact Nutek For A Possible Solution.'),(sAlmText:='File Create Error While Editing',sRcyText:='An Error Was Encountered While Trying To Create File. Please Contact Nutek For A Possible Solution.'),(sAlmText:='File Write Error While Editing',sRcyText:='An Error Was Encountered While Trying To Write File. Please Contact Nutek For A Possible Solution.'),(sAlmText:='File Close Error While Editing',sRcyText:='An Error Was Encountered While Trying To Close File. Please Contact Nutek For A Possible Solution.'),(sAlmText:='Directory Does Not Exist While Editing',sRcyText:='The Directory Does Not Exist.Please Contact Nutek For A Possible Solution.'),(sAlmText:='File Open Error While Loading Current Recipe',sRcyText:='An Error Was Encountered While Trying To Open File. Please Contact Nutek For A Possible Solution.'),(sAlmText:='File Create Error While Loading Current Recipe',sRcyText:='An Error Was Encountered While Trying To Create File. Please Contact Nutek For A Possible Solution.'),(sAlmText:='File Write Error While Loading Current Recipe',sRcyText:='An Error Was Encountered While Trying To Write File. Please Contact Nutek For A Possible Solution.'),(sAlmText:='File Close Error While Loading Current Recipe',sRcyText:='An Error Was Encountered While Trying To Close File. Please Contact Nutek For A Possible Solution.'),(sAlmText:='Directory Does Not Exist While Loading Current Recipe',sRcyText:='The Directory Does Not Exist.Please Contact Nutek For A Possible Solution.'),(sAlmText:='File Open Error While Reading Current Recipe',sRcyText:='An Error Was Encountered While Trying To Open File. Please Contact Nutek For A Possible Solution.'),(sAlmText:='File Read Error While Reading Current Recipe',sRcyText:='An Error Was Encountered While Trying To Read File. Please Contact Nutek For A Possible Solution.'),(sAlmText:='File Close Error While Reading Current Recipe',sRcyText:='An Error Was Encountered While Trying To Close File. Please Contact Nutek For A Possible Solution.'),(sAlmText:='File Open Error While Writing Current Recipe Parameter',sRcyText:='An Error Was Encountered While Trying To Open File. Please Contact Nutek For A Possible Solution.'),(sAlmText:='File Create Error While Writing Current Recipe Parameter',sRcyText:='An Error Was Encountered While Trying To Create File. Please Contact Nutek For A Possible Solution.'),(sAlmText:='File Write Error While Writing Current Recipe Parameter',sRcyText:='An Error Was Encountered While Trying To Write File. Please Contact Nutek For A Possible Solution.'),(sAlmText:='File Close Error While Writing Current Recipe Parameter',sRcyText:='An Error Was Encountered While Trying To Close File. Please Contact Nutek For A Possible Solution.'),(sAlmText:='Directory Does Not Exist While Writing Current Recipe Parameter',sRcyText:='The Directory Does Not Exist.Please Contact Nutek For A Possible Solution.'),(sAlmText:='File Open Error While Writing Saving List',sRcyText:='An Error Was Encountered While Trying To Open File. Please Contact Nutek For A Possible Solution.'),(sAlmText:='File Create Error While Writing Saving List',sRcyText:='An Error Was Encountered While Trying To Create File. Please Contact Nutek For A Possible Solution.'),(sAlmText:='File Write Error While Writing Saving List',sRcyText:='An Error Was Encountered While Trying To Write File. Please Contact Nutek For A Possible Solution.'),(sAlmText:='File Close Error While Writing Saving List',sRcyText:='An Error Was Encountered While Trying To Close File. Please Contact Nutek For A Possible Solution.'),(sAlmText:='Directory Does Not Exist While Writing Saving List',sRcyText:='The Directory Does Not Exist.Please Contact Nutek For A Possible Solution.'),57(0)];
END_VAR
(**)
(*Local Output*)
VAR
	bNmExist : BOOL;
	bNmNotExist : BOOL;
	bNmEmpty : BOOL;
	bListFull : BOOL;
	sDebug : STRING[300];
	tyTempRecipe : tyProdRcpParam;
	a_tyCurrList : ARRAY[1..c_udiProdRcpMax] OF tyProdRcpParam;
	a_tyFilterList : ARRAY[1..c_udiProdRcpMax] OF tyProdRcpParam;
	a_tySortList : ARRAY[1..c_udiProdRcpMax] OF tyProdRcpParam;
	a_tyScanList : ARRAY[1..c_udiProdRcpMax] OF tyProdRcpParam;
	tyInfoOut : tyProdRcpParam;
	bFileNotFound : BOOL;
	a_tyCurrRcp : ARRAY[0..5] OF tyProdRcpParam;
	iFilterCtr : INT;
END_VAR
(**)
(*Local Input*)
VAR
	udiRstErr : UDINT := 0;
	dtCurrDT : DATE_AND_TIME;
	sSearch : STRING[254] := '';
	sScan : STRING[254] := '';
	tyInfoIn : tyProdRcpParam;
	tyCurrRcpWr : tyProdRcpParam;
	sListFileName : STRING[80] := 'ProductRecipeList.dat';
	sSingleFileName : STRING[80] := 'ProductRecipe.dat';
	sProgNm : STRING[15] := 'ProdRcp';
	bNtSettingsLoadDone : BOOL := TRUE;
	bWidth2Prep : BOOL;
	uiSortNo : UDINT := 0;
END_VAR
(**)
(*Local*)
VAR
	sEndRcpName : STRING[254];
	bCreateRcp : BOOL;
	udiSortCurrenTotalCntr : UDINT;
	iSortCurrentInnerCntr : INT;
	iSortCurrentOuterCntr : INT;
	iTotalRcp : INT;
	udi : UDINT;
	bRstErr : BOOL;
	udiRstErrOld : UDINT;
	bInitDone : BOOL;
	bInitialDone : BOOL;
	usiStep : USINT;
	udiAddStatus : UDINT;
	a_tyListTemp : ARRAY[1..c_udiProdRcpMax] OF tyProdRcpParam;
	fbDirCreate1 : fbDirCreate;
	fbDirCreate2 : fbDirCreate;
	fbFileReadList : fbFileFullRead;
	fbFileWriteList : fbFileFullWrite;
	fbFileReadSingle : fbFileFullRead;
	fbFileWriteSingle : fbFileFullWrite;
	fbFileLoadSingle : fbFileFullWrite;
	udiModuleNum : UDINT := 4801;
END_VAR
```

#### Act_Alarm.st
```iecst
(** 2019-03-25 **)
ACTION Act_Alarm:

	//Error
	IF EDGEPOS(eStatus = Error) THEN

		tyAlmData.sProgNm		:= p_sProgNm;
		tyAlmData.udiCode		:= udiStatus;
		tyAlmData.eSeverity		:= AlmSeverityError;
		tyAlmData.udiRunTime	:= tyAlmData.udiRunTime + 1;
		tyAlmData.bAlm			:= TRUE;
		tyAlmData.udiModuleNum  := udiModuleNum;
		g_sProdRcpProgNm		:= p_sProgNm;
		//Get Error Message
		IF tyAlmData.udiCode < 10000 OR tyAlmData.udiCode > 10099 THEN
			tyAlmData.sAlmMsg	:= 'Unknown';
			tyAlmData.sRcyMsg	:= 'Unknown';
		ELSE
			tyAlmData.sAlmMsg	:= a_tyAlmText[tyAlmData.udiCode].sAlmText;
			tyAlmData.sRcyMsg	:= a_tyAlmText[tyAlmData.udiCode].sRcyText;
		END_IF

		sStatTxt	:= tyAlmData.sAlmMsg;

	ELSIF bRstErr AND (tyAlmData.udiCode <> 0) THEN

		tyAlmData.udiCode	:= 0;
		tyAlmData.eSeverity	:= AlmSeverityNA;
		tyAlmData.sAlmMsg	:= '';
		tyAlmData.sRcyMsg	:= '';
		tyAlmData.bAlm		:= FALSE;
		sStatTxt	:= a_sStatText[eStat];

	END_IF

END_ACTION
```

#### Act_InitGlobal.st
```iecst
(** 2020-06-08 **)
ACTION Act_InitGlobal:

	(* Always Change If Project Change *)

	//Pass Data To Link
	p_bLinkStartupRun ACCESS p_StartupRun;
	p_bLinkNtParamLCSManageRcpPrep ACCESS p_NtParamLCSManageRcpPrep;
	p_bLinkMcParamLCSManageRcpEn ACCESS p_McParamLCSManageRcpEn;
	p_eLinkLCSMngRcpProdRcpAct ACCESS p_LCSMngRcpProdRcpAct;
	p_eLinkUIProdRcpAct ACCESS p_UIProdRcpAct;
	p_eLinkMag ACCESS p_NtParamProjMag;
	//Pass Data To Internal Use
	p_udiRstErr ACCESS p_RstErrReset;
	p_dtCurrDT ACCESS p_TimeCurrDT;
	p_sSearch ACCESS p_UIProdRcpSearch;
	p_tyInfoIn ACCESS p_UIProdRcpInfoIn;
	p_tyCurrRcpWr ACCESS p_UIProdRcpCurrRcpWr;
	p_sListFileName ACCESS p_NtParamProdRcpListFileNm;
	p_sSingleFileName ACCESS p_NtParamProdRcpSingleFileNm;
	p_sProgNm ACCESS p_NtParamProdRcpProgNm;
	p_bNtSettingsLoadDone ACCESS p_StartupNtSettingsLoadDone;
	p_bWidth2Prep ACCESS p_NtParamLFWidth2Prep;
	(* Always Change If Project Change *)

END_ACTION
```

#### Act_Link.st
```iecst
(** 2019-04-30 **)
ACTION Act_Link:

	IF (p_eAct = ProdRcpActAddEdit) OR (p_eAct = ProdRcpActAdd) OR (p_eAct = ProdRcpActEdit) THEN

		rWidthInMM				:= DINT_TO_REAL(p_tyInfoIn.diWidthInUM);
		rWidthInMM2				:= DINT_TO_REAL(p_tyInfoIn.diWidthInUM2);
		rWidthInMM				:= rWidthInMM / 1000;
		rWidthInMM2				:= rWidthInMM2 / 1000;
		sWidthInMM				:= REAL_TO_STRING(rWidthInMM);
		sWidthInMM2				:= REAL_TO_STRING(rWidthInMM2);

		rWidthInMMRear				:= DINT_TO_REAL(p_tyInfoIn.diWidthInUMRear);
		rWidthInMMRear				:= rWidthInMMRear / 1000;
		sWidthInMMRear				:= REAL_TO_STRING(rWidthInMMRear);

		IF p_bWidth2Prep THEN
			p_tyInfoIn.sDisplayInfo	:= sWidthInMM;
			p_tyInfoIn.sDisplayInfo	:= CONCAT(p_tyInfoIn.sDisplayInfo , ' | ');
			p_tyInfoIn.sDisplayInfo	:= CONCAT(p_tyInfoIn.sDisplayInfo , sWidthInMM2);
			p_tyInfoIn.sDisplayInfo	:= CONCAT(p_tyInfoIn.sDisplayInfo , ' mm');
		ELSIF p_eLinkMag = LDMagQuadruple THEN
			p_tyInfoIn.sDisplayInfo	:= sWidthInMM;
			p_tyInfoIn.sDisplayInfo	:= CONCAT(p_tyInfoIn.sDisplayInfo , ' | ');
			p_tyInfoIn.sDisplayInfo	:= CONCAT(p_tyInfoIn.sDisplayInfo , sWidthInMMRear);
			p_tyInfoIn.sDisplayInfo	:= CONCAT(p_tyInfoIn.sDisplayInfo , ' mm');

		ELSE
			p_tyInfoIn.sDisplayInfo	:= sWidthInMM;
			p_tyInfoIn.sDisplayInfo	:= CONCAT(p_tyInfoIn.sDisplayInfo , ' mm');
		END_IF

	END_IF

END_ACTION
```

#### Act_Main.st
```iecst
(** 2020-06-08 **)
ACTION Act_Main:

	//Main
	CASE eStat OF

		ProdRcpActIdle:
			IF eStatus <> Idle THEN	//Reset Data
				//Private
				fbDirCreate1(bEn := FALSE);
				fbDirCreate2(bEn := FALSE);
				fbFileReadList(bEn := FALSE);
				fbFileWriteList(bEn := FALSE);
				fbFileReadSingle(bEn := FALSE);
				fbFileWriteSingle(bEn := FALSE);
				fbFileLoadSingle(bEn := FALSE);
				usiStep				:= 0;
				udiAddStatus		:= 0;

				bNmExist		:= FALSE;
				bNmNotExist		:= FALSE;
				bNmEmpty		:= FALSE;
				bListFull		:= FALSE;
				bFileNotFound	:= FALSE;
				iTotalRcp 		:= 0;

				memset(ADR(tyTempRecipe), 0 , SIZEOF(tyTempRecipe));

				sStatTxt	:= a_sStatText[eStat];

			END_IF

			eStatus	:= Idle;

		ProdRcpActCreateDir:
			IF eStatus = Idle OR eStatus = Busy THEN

				eStatus	:= Busy;

				sStatTxt	:= a_sStatText[eStat];

				CASE usiStep OF
					0:
						fbDirCreate1(bEn := TRUE);
						IF fbDirCreate1.udiStatus = 0 THEN
							usiStep	:= 1;
						ELSIF fbDirCreate1.udiStatus < 65534 THEN
							eStatus		:= Error;

							IF fbDirCreate1.udiStatus = 1908 THEN
								udiStatus	:= 10000;	//Create User Directory Error
							ELSE
								udiStatus	:= fbDirCreate1.udiStatus;
							END_IF
						END_IF

					1:
						fbDirCreate2(bEn := TRUE);
						IF fbDirCreate2.udiStatus = 0 THEN
							eStatus	:= Done;
						ELSIF fbDirCreate2.udiStatus < 65534 THEN
							eStatus		:= Error;

							IF fbDirCreate2.udiStatus = 1908 THEN
								udiStatus	:= 10001;	//Create Product Recipe Directory Error
							ELSE
								udiStatus	:= fbDirCreate2.udiStatus;
							END_IF
						END_IF

				END_CASE

			END_IF

		ProdRcpActAddEdit:
			IF eStatus = Idle OR eStatus = Busy THEN

				eStatus	:= Busy;

				sStatTxt	:= a_sStatText[eStat];

				CASE usiStep OF
					0:	//Edit Recipe
						udiAddStatus	:= fRecipeAddEdit(ADR(p_tyInfoIn) , ADR(a_tyListTemp) , SIZEOF(a_tyListTemp[1]) , ADR(a_tyListTemp[1].sRcpNm) , SIZEOF(a_tyListTemp[1].sRcpNm) , p_udiMax);

						IF udiAddStatus = 1600 THEN	//Recipe Name Empty
							bNmEmpty	:= TRUE;
							eStatus		:= Done;

						ELSIF udiAddStatus = 1601 THEN	//Recipe Full
							bListFull	:= TRUE;
							eStatus		:= Done;

						ELSIF udiAddStatus = 0 THEN	//OK
							usiStep	:= 1;

						END_IF

					1:	//Write Into File
						fbFileWriteList(bEn := TRUE);

						IF fbFileWriteList.udiStatus = 0 THEN
							a_tyCurrList	:= a_tyListTemp;

							eStatus := Done;

						ELSIF fbFileWriteList.udiStatus < 65534 THEN
							a_tyListTemp	:= a_tyCurrList;
							eStatus			:= Error;

							IF fbFileWriteList.udiStatus = 1900 THEN
								udiStatus	:= 10002;	//File Open Error While Adding & Editing
							ELSIF fbFileWriteList.udiStatus = 1901 THEN
								udiStatus	:= 10003;	//File Create Error While Adding & Editing
							ELSIF fbFileWriteList.udiStatus = 1903 THEN
								udiStatus	:= 10004;	//File Write Error While Adding & Editing
							ELSIF fbFileWriteList.udiStatus = 1904 THEN
								udiStatus	:= 10005;	//File Close Error While Adding & Editing
							ELSIF fbFileWriteList.udiStatus = 1914 THEN
								udiStatus	:= 10013;	//Directory Does Not Exist While Adding & Editing
							ELSE
								udiStatus	:= fbFileWriteList.udiStatus;
							END_IF
						END_IF

				END_CASE

			END_IF

		ProdRcpActDel:
			IF eStatus = Idle OR eStatus = Busy THEN

				eStatus	:= Busy;

				sStatTxt	:= a_sStatText[eStat];

				CASE usiStep OF
					0:	//Edit User
						udiAddStatus	:= fRecipeDelete(ADR(p_tyInfoIn) , ADR(a_tyListTemp) , SIZEOF(a_tyListTemp[1]) , ADR(a_tyListTemp[1].sRcpNm) , SIZEOF(a_tyListTemp[1].sRcpNm) , p_udiMax);

						IF udiAddStatus = 1600 THEN	//Recipe Name Empty
							bNmEmpty	:= TRUE;
							eStatus		:= Done;

						ELSIF udiAddStatus = 1603 THEN	//Recipe Not Exist
							bNmNotExist	:= TRUE;
							eStatus		:= Done;

						ELSIF udiAddStatus = 0 THEN	//OK
							usiStep	:= 1;

						END_IF

					1:	//Write Into File
						fbFileWriteList(bEn := TRUE);

						IF fbFileWriteList.udiStatus = 0 THEN
							a_tyCurrList	:= a_tyListTemp;
							eStatus := Done;

						ELSIF fbFileWriteList.udiStatus < 65534 THEN
							a_tyListTemp	:= a_tyCurrList;
							eStatus			:= Error;

							IF fbFileWriteList.udiStatus = 1900 THEN
								udiStatus	:= 10006;	//File Open Error While Deleting
							ELSIF fbFileWriteList.udiStatus = 1901 THEN
								udiStatus	:= 10007;	//File Create Error While Deleting
							ELSIF fbFileWriteList.udiStatus = 1903 THEN
								udiStatus	:= 10008;	//File Write Error While Deleting
							ELSIF fbFileWriteList.udiStatus = 1904 THEN
								udiStatus	:= 10009;	//File Close Error While Deleting
							ELSIF fbFileWriteList.udiStatus = 1914 THEN
								udiStatus	:= 10014;	//Directory Does Not Exist While Deleting
							ELSE
								udiStatus	:= fbFileWriteList.udiStatus;
							END_IF

						END_IF

				END_CASE

			END_IF

		ProdRcpActGetInfo:
			IF eStatus = Idle OR eStatus = Busy THEN

				sStatTxt	:= a_sStatText[eStat];

				IF p_tyInfoIn.sRcpNm = '' THEN
					bNmEmpty	:= TRUE;
					bNmNotExist	:= TRUE;
				ELSE
					bNmNotExist	:= (fRecipeGetInfo(p_tyInfoIn.sRcpNm , ADR(tyInfoOut) , ADR(a_tyCurrList) , SIZEOF(a_tyCurrList[1]) , ADR(a_tyCurrList[1].sRcpNm) , SIZEOF(a_tyCurrList[1].sRcpNm) , p_udiMax)) = 0;
				END_IF

				eStatus	:= Done;

			END_IF

		ProdRcpActGetList:
			IF eStatus = Idle OR eStatus = Busy THEN

				eStatus	:= Busy;

				sStatTxt	:= a_sStatText[eStat];

				fbFileReadList(bEn := TRUE);

				IF fbFileReadList.udiStatus = 0 THEN
					a_tyListTemp	:= a_tyCurrList;
					eStatus			:= Done;

				ELSIF fbFileReadList.udiStatus < 65534 THEN
					eStatus		:= Error;

					IF fbFileReadList.udiStatus = 1900 THEN
						udiStatus	:= 10010;	//File Open Error While Getting List
					ELSIF fbFileReadList.udiStatus = 1902 THEN
						udiStatus	:= 10011;	//File Read Error While Getting List
					ELSIF fbFileReadList.udiStatus = 1904 THEN
						udiStatus	:= 10012;	//File Close Error While Getting List
					ELSIF fbFileReadList.udiStatus = 1915 THEN
						eStatus			:= Done;
						bFileNotFound	:= TRUE;
					ELSE
						udiStatus	:= fbFileReadList.udiStatus;
					END_IF

				END_IF

			END_IF

		ProdRcpActFilter:

			IF eStatus = Idle OR eStatus = Busy THEN

				eStatus := Busy;

				sStatTxt	:= a_sStatText[eStat];

				CASE usiStep OF
					0:
						fRecipeFilter(p_sSearch , ADR(a_tyFilterList) , ADR(a_tyCurrList) , SIZEOF(a_tyCurrList[1]) , ADR(a_tyCurrList[1].sRcpNm) ,
						SIZEOF(a_tyCurrList[1].sRcpNm) , p_udiMax, 0, 499, iFilterCtr);
						usiStep := 1;
					1:
						fRecipeFilter(p_sSearch , ADR(a_tyFilterList) , ADR(a_tyCurrList) , SIZEOF(a_tyCurrList[1]) , ADR(a_tyCurrList[1].sRcpNm) ,
						SIZEOF(a_tyCurrList[1].sRcpNm) , p_udiMax, 500, 999, iFilterCtr);
						usiStep := 2;
					2:
						fRecipeFilter(p_sSearch , ADR(a_tyFilterList) , ADR(a_tyCurrList) , SIZEOF(a_tyCurrList[1]) , ADR(a_tyCurrList[1].sRcpNm) ,
						SIZEOF(a_tyCurrList[1].sRcpNm) , p_udiMax, 1000, 1499, iFilterCtr);
						usiStep := 3;
					3:
						fRecipeFilter(p_sSearch , ADR(a_tyFilterList) , ADR(a_tyCurrList) , SIZEOF(a_tyCurrList[1]) , ADR(a_tyCurrList[1].sRcpNm) ,
						SIZEOF(a_tyCurrList[1].sRcpNm) , p_udiMax, 1500, 1999, iFilterCtr);
						eStatus := Done;

				END_CASE

			END_IF;

		ProdRcpActLoadRcp:
			IF eStatus = Idle OR eStatus = Busy THEN

				sStatTxt	:= a_sStatText[eStat];

				CASE usiStep OF
					0:	//Get Current Recipe
						IF p_tyInfoIn.sRcpNm = '' THEN
							bNmEmpty	:= TRUE;
							bNmNotExist	:= TRUE;

							eStatus	:= Done;
						ELSE
							bNmNotExist	:= (fRecipeGetInfo(p_tyInfoIn.sRcpNm , ADR(a_tyCurrRcp[0]) , ADR(a_tyCurrList) , SIZEOF(a_tyCurrList[1]) , ADR(a_tyCurrList[1].sRcpNm) , SIZEOF(a_tyCurrList[1].sRcpNm) , p_udiMax)) = 0;

							IF bNmNotExist = TRUE THEN
								eStatus	:= Done;
							ELSE
								usiStep	:= 1;
							END_IF

						END_IF

					1:	//Write Into File
						fbFileLoadSingle(bEn := TRUE);

						IF fbFileLoadSingle.udiStatus = 0 THEN
							eStatus			:= Done;
						ELSIF fbFileLoadSingle.udiStatus < 65534 THEN
							eStatus			:= Error;

							IF fbFileLoadSingle.udiStatus = 1900 THEN
								udiStatus	:= 10025;	//File Open Error While Loading Current Recipe
							ELSIF fbFileLoadSingle.udiStatus = 1901 THEN
								udiStatus	:= 10026;	//File Create Error While Loading Current Recipe
							ELSIF fbFileLoadSingle.udiStatus = 1903 THEN
								udiStatus	:= 10027;	//File Write Error While Loading Current Recipe
							ELSIF fbFileLoadSingle.udiStatus = 1904 THEN
								udiStatus	:= 10028;	//File Close Error While Loading Current Recipe
							ELSIF fbFileLoadSingle.udiStatus = 1914 THEN
								udiStatus	:= 10029;	//Directory Does Not Exist While Loading Current Recipe
							ELSE
								udiStatus	:= fbFileLoadSingle.udiStatus;
							END_IF
						END_IF

				END_CASE

			END_IF

		ProdRcpActAdd:
			IF eStatus = Idle OR eStatus = Busy THEN

				eStatus	:= Busy;

				sStatTxt	:= a_sStatText[eStat];

				CASE usiStep OF
					0:	//Edit Recipe
						udiAddStatus	:= fRecipeAdd(ADR(p_tyInfoIn) , ADR(a_tyListTemp) , SIZEOF(a_tyListTemp[1]) , ADR(a_tyListTemp[1].sRcpNm) , SIZEOF(a_tyListTemp[1].sRcpNm) , p_udiMax);

						IF udiAddStatus = 1600 THEN	//Recipe Name Empty
							bNmEmpty	:= TRUE;
							eStatus		:= Done;

						ELSIF udiAddStatus = 1601 THEN	//Recipe Full
							bListFull	:= TRUE;
							eStatus		:= Done;

						ELSIF udiAddStatus = 1602 THEN	//Recipe Name Exist
							bNmExist	:= TRUE;
							eStatus		:= Done;

						ELSIF udiAddStatus = 0 THEN	//OK
							usiStep	:= 1;

						END_IF

					1:	//Write Into File
						fbFileWriteList(bEn := TRUE);

						IF fbFileWriteList.udiStatus = 0 THEN
							a_tyCurrList	:= a_tyListTemp;
							eStatus			:= Done;

						ELSIF fbFileWriteList.udiStatus < 65534 THEN
							a_tyListTemp	:= a_tyCurrList;
							eStatus			:= Error;

							IF fbFileWriteList.udiStatus = 1900 THEN
								udiStatus	:= 10015;	//File Open Error While Adding
							ELSIF fbFileWriteList.udiStatus = 1901 THEN
								udiStatus	:= 10016;	//File Create Error While Adding
							ELSIF fbFileWriteList.udiStatus = 1903 THEN
								udiStatus	:= 10017;	//File Write Error While Adding
							ELSIF fbFileWriteList.udiStatus = 1904 THEN
								udiStatus	:= 10018;	//File Close Error While Adding
							ELSIF fbFileWriteList.udiStatus = 1914 THEN
								udiStatus	:= 10019;	//Directory Does Not Exist While Adding
							ELSE
								udiStatus	:= fbFileWriteList.udiStatus;
							END_IF
						END_IF
				END_CASE

			END_IF

		ProdRcpActEdit:
			IF eStatus = Idle OR eStatus = Busy THEN

				eStatus	:= Busy;

				sStatTxt	:= a_sStatText[eStat];

				CASE usiStep OF
					0:	//Edit Recipe
						udiAddStatus	:= fRecipeEdit(ADR(p_tyInfoIn) , ADR(a_tyListTemp) , SIZEOF(a_tyListTemp[1]) , ADR(a_tyListTemp[1].sRcpNm) , SIZEOF(a_tyListTemp[1].sRcpNm) , p_udiMax);

						IF udiAddStatus = 1600 THEN	//Recipe Name Empty
							bNmEmpty	:= TRUE;
							eStatus		:= Done;

						ELSIF udiAddStatus = 1603 THEN	//Recipe Not Exist
							bNmNotExist	:= TRUE;
							eStatus		:= Done;

						ELSIF udiAddStatus = 0 THEN	//OK
							usiStep	:= 1;

						END_IF

					1:	//Write Into File
						fbFileWriteList(bEn := TRUE);

						IF fbFileWriteList.udiStatus = 0 THEN
							a_tyCurrList	:= a_tyListTemp;
							eStatus			:= Done;

						ELSIF fbFileWriteList.udiStatus < 65534 THEN
							a_tyListTemp	:= a_tyCurrList;
							eStatus			:= Error;

							IF fbFileWriteList.udiStatus = 1900 THEN
								udiStatus	:= 10020;	//File Open Error While Adding & Editing
							ELSIF fbFileWriteList.udiStatus = 1901 THEN
								udiStatus	:= 10021;	//File Create Error While Adding & Editing
							ELSIF fbFileWriteList.udiStatus = 1903 THEN
								udiStatus	:= 10022;	//File Write Error While Adding & Editing
							ELSIF fbFileWriteList.udiStatus = 1904 THEN
								udiStatus	:= 10023;	//File Close Error While Adding & Editing
							ELSIF fbFileWriteList.udiStatus = 1914 THEN
								udiStatus	:= 10024;	//Directory Does Not Exist While Adding & Editing
							ELSE
								udiStatus	:= fbFileWriteList.udiStatus;
							END_IF
						END_IF

				END_CASE

			END_IF

		ProdRcpActReadCurrRcp:
			IF eStatus = Idle OR eStatus = Busy THEN

				eStatus	:= Busy;

				sStatTxt	:= a_sStatText[eStat];

				fbFileReadSingle(bEn := TRUE);
				IF fbFileReadSingle.udiStatus = 0 THEN
					eStatus			:= Done;

				ELSIF fbFileReadSingle.udiStatus < 65534 THEN
					eStatus		:= Error;

					IF fbFileReadSingle.udiStatus = 1900 THEN
						udiStatus	:= 10030;	//File Open Error While Reading Current Recipe
					ELSIF fbFileReadSingle.udiStatus = 1902 THEN
						udiStatus	:= 10031;	//File Read Error While Reading Current Recipe
					ELSIF fbFileReadSingle.udiStatus = 1904 THEN
						udiStatus	:= 10032;	//File Close Error While Reading Current Recipe
					ELSIF fbFileReadSingle.udiStatus = 1915 THEN
						eStatus			:= Done;
						bFileNotFound	:= TRUE;
					ELSE
						udiStatus	:= fbFileReadSingle.udiStatus;
					END_IF
				END_IF

			END_IF

		ProdRcpActWriteCurrRcpParam:
			IF eStatus = Idle OR eStatus = Busy THEN

				sStatTxt	:= a_sStatText[eStat];

				fbFileWriteSingle(bEn := TRUE);

				IF fbFileWriteSingle.udiStatus = 0 THEN
					a_tyCurrRcp[0]	:= p_tyCurrRcpWr;
					eStatus			:= Done;
				ELSIF fbFileWriteSingle.udiStatus < 65534 THEN
					eStatus			:= Error;

					IF fbFileWriteSingle.udiStatus = 1900 THEN
						udiStatus	:= 10033;	//File Open Error While Writing Current Recipe Parameter
					ELSIF fbFileWriteSingle.udiStatus = 1901 THEN
						udiStatus	:= 10034;	//File Create Error While Writing Current Recipe Parameter
					ELSIF fbFileWriteSingle.udiStatus = 1903 THEN
						udiStatus	:= 10035;	//File Write Error While Writing Current Recipe Parameter
					ELSIF fbFileWriteSingle.udiStatus = 1904 THEN
						udiStatus	:= 10036;	//File Close Error While Writing Current Recipe Parameter
					ELSIF fbFileWriteSingle.udiStatus = 1914 THEN
						udiStatus	:= 10037;	//Directory Does Not Exist Writing Current Recipe Parameter
					ELSE
						udiStatus	:= fbFileWriteSingle.udiStatus;
					END_IF
				END_IF

			END_IF

		ProdRcpActSaveList:
			IF eStatus = Idle OR eStatus = Busy THEN

				eStatus	:= Busy;

				sStatTxt	:= a_sStatText[eStat];

				CASE usiStep OF

					0:
						a_tyListTemp	:= a_tyCurrList;

						fbFileWriteList(bEn := TRUE);

						IF fbFileWriteList.udiStatus = 0 THEN
							eStatus			:= Done;

						ELSIF fbFileWriteList.udiStatus < 65534 THEN
							eStatus			:= Error;

							IF fbFileWriteList.udiStatus = 1900 THEN
								udiStatus	:= 10038;	//File Open Error While Saving List
							ELSIF fbFileWriteList.udiStatus = 1901 THEN
								udiStatus	:= 10039;	//File Create Error While Saving List
							ELSIF fbFileWriteList.udiStatus = 1903 THEN
								udiStatus	:= 10040;	//File Write Error While Saving List
							ELSIF fbFileWriteList.udiStatus = 1904 THEN
								udiStatus	:= 10041;	//File Close Error While Saving List
							ELSIF fbFileWriteList.udiStatus = 1914 THEN
								udiStatus	:= 10042;	//Directory Does Not Exist While Saving List
							ELSE
								udiStatus	:= fbFileWriteList.udiStatus;
							END_IF
						END_IF

				END_CASE

			END_IF

		ProdRcpActSort:
			IF eStatus = Idle OR eStatus = Busy THEN

				sStatTxt	:= a_sStatText[eStat];

				CASE usiStep OF

					0:

						FOR udi := 1 TO c_udiProdRcpMax DO
							IF p_sSearch <> '' THEN
								IF a_tyFilterList[udi].sRcpNm = '' THEN
									usiStep := 1;
									EXIT;
								ELSIF udi = c_udiProdRcpMax THEN
									iTotalRcp := UDINT_TO_INT(c_udiProdRcpMax);
									usiStep := 1;
									EXIT;
								ELSE
									iTotalRcp := iTotalRcp +1;
								END_IF
							ELSE
								IF a_tyCurrList[udi].sRcpNm = '' THEN
									usiStep := 1;
									EXIT;
								ELSIF udi = c_udiProdRcpMax THEN
									iTotalRcp := UDINT_TO_INT(c_udiProdRcpMax);
									usiStep := 1;
									EXIT;
								ELSE
									iTotalRcp := iTotalRcp +1;
								END_IF
							END_IF
						END_FOR

					1:
						IF p_sSearch <> '' THEN
							memcpy(ADR(a_tySortList),ADR(a_tyFilterList), SIZEOF(a_tyFilterList));
						ELSE
							memcpy(ADR(a_tySortList),ADR(a_tyCurrList), SIZEOF(a_tyCurrList));
						END_IF

						iSortCurrentOuterCntr	:= 0;
						iSortCurrentInnerCntr	:= 1 ;

						udiSortCurrenTotalCntr	:= 0;

						usiStep := 2;

					2:

						IF iSortCurrentOuterCntr < iTotalRcp THEN

							FOR iSortCurrentInnerCntr:= iSortCurrentOuterCntr+1 TO iTotalRcp-1 DO

								IF fRecipeNmCompare(ADR(a_tySortList[iSortCurrentOuterCntr+1].sRcpNm),ADR(a_tySortList[iSortCurrentInnerCntr+1].sRcpNm),SIZEOF(a_tySortList[1].sRcpNm),ADR(sDebug)) THEN

									memcpy(ADR(tyTempRecipe), ADR(a_tySortList[iSortCurrentOuterCntr+1]), SIZEOF(a_tySortList[1]));
									memcpy(ADR(a_tySortList[iSortCurrentOuterCntr+1]), ADR(a_tySortList[iSortCurrentInnerCntr+1]), SIZEOF(a_tySortList[1]));
									memcpy(ADR(a_tySortList[iSortCurrentInnerCntr+1]), ADR(tyTempRecipe), SIZEOF(a_tySortList[1]));

								END_IF

								udiSortCurrenTotalCntr	:= udiSortCurrenTotalCntr + 1;

							END_FOR

							iSortCurrentOuterCntr	:= iSortCurrentOuterCntr + 1;

						ELSE
							usiStep := 3;
						END_IF

					3:
						eStatus	:= Done;

				END_CASE

			END_IF

		ProdRcpActEndCharFilter:
			IF eStatus = Idle OR eStatus = Busy THEN

				sStatTxt	:= a_sStatText[eStat];

				fRecipeLastCharFilter(p_sScan , ADR(a_tyScanList) , ADR(a_tyCurrList) , SIZEOF(a_tyCurrList[1]) , ADR(a_tyCurrList[1].sRcpNm) , SIZEOF(a_tyCurrList[1].sRcpNm) , p_udiMax);

				eStatus	:= Done;

			END_IF

	END_CASE

END_ACTION
```

#### Init.st
```iecst
(** 2020-06-08 **)
PROGRAM _INIT

	(* Always Change If Project Change *)

	//Pass Address To Global Address For External Use
	//Action, State & Status
	p_ProdRcpStat		:= ADR(eStat);
	p_ProdRcpStatus		:= ADR(eStatus);
	p_ProdRcpStatTxt	:= ADR(sStatTxt);

	//Alarm
	p_ProdRcpAlmData	:= ADR(tyAlmData);

	//Output
	p_ProdRcpNmExist		:= ADR(bNmExist);
	p_ProdRcpNmNotExist		:= ADR(bNmNotExist);
	p_ProdRcpNmEmpty		:= ADR(bNmEmpty);
	p_ProdRcpListFull		:= ADR(bListFull);
	p_ProdRcpCurrList		:= ADR(a_tyCurrList);
	p_ProdRcpFilterList		:= ADR(a_tyFilterList);
	p_ProdRcpSortedList		:= ADR(a_tySortList);
	p_ProdRcpScanList		:= ADR(a_tyScanList);
	p_ProdRcpInfoOut		:= ADR(tyInfoOut);
	p_ProdRcpFileNotFound	:= ADR(bFileNotFound);
	p_ProdRcpCurrRcpAll		:= ADR(a_tyCurrRcp);

	p_ProdRcpCurrRcp0				:= ADR(a_tyCurrRcp[0]);
	p_ProdRcpCurrRcp0Nm				:= ADR(a_tyCurrRcp[0].sRcpNm);
	p_ProdRcpCurrRcp0Width			:= ADR(a_tyCurrRcp[0].diWidthInUM);
	p_ProdRcpCurrRcp0MinSltValue	:= ADR(a_tyCurrRcp[0].diMinSltValue);
	p_ProdRcpCurrRcp0MaxSltValue	:= ADR(a_tyCurrRcp[0].diMaxSltValue);
	p_ProdRcpCurrRcp0Pitch			:= ADR(a_tyCurrRcp[0].diPitch);
	p_ProdRcpCurrRcp0McMod			:= ADR(a_tyCurrRcp[0].usiMcMod);
	p_ProdRcpCurrRcp0FlippedBrd		:= ADR(a_tyCurrRcp[0].usiFlippedBrd);
	p_ProdRcpCurrRcp0TopToBtm		:= ADR(a_tyCurrRcp[0].bTopToBtm);
	p_ProdRcpCurrRcp0LongBrd		:= ADR(a_tyCurrRcp[0].bLongBrd);
	p_ProdRcpCurrRcp0DisplayInfo	:= ADR(a_tyCurrRcp[0].sDisplayInfo);
	p_ProdRcpCurrRcp0LastModified	:= ADR(a_tyCurrRcp[0].dtLastModified);
	p_ProdRcpCurrRcp0Width2 		:= ADR(a_tyCurrRcp[0].diWidthInUM2);
	p_ProdRcpCurrRcp0WidthRear		:= ADR(a_tyCurrRcp[0].diWidthInUMRear);
	p_ProdRcpCurrRcp0PitchRear		:= ADR(a_tyCurrRcp[0].diPitchRear);
	p_ProdRcpCurrRcp0MinSltRear		:= ADR(a_tyCurrRcp[0].diMinSltValueRear);
	p_ProdRcpCurrRcp0MaxSltRear		:= ADR(a_tyCurrRcp[0].diMaxSltValueRear);
	p_ProdRcpCurrRcp0PshrOffset		:= ADR(a_tyCurrRcp[0].diPshrOffset);
	p_ProdRcpCurrRcp0MtrPshrExtSpd	:= ADR(a_tyCurrRcp[0].diMtrPshrExtSpd);
	p_ProdRcpCurrRcp0MtrPshrExtTorq	:= ADR(a_tyCurrRcp[0].diMtrPshrExtTorq);

	p_ProdRcpCurrRcp1				:= ADR(a_tyCurrRcp[1]);
	p_ProdRcpCurrRcp1Nm				:= ADR(a_tyCurrRcp[1].sRcpNm);
	p_ProdRcpCurrRcp1Width			:= ADR(a_tyCurrRcp[1].diWidthInUM);
	p_ProdRcpCurrRcp1MinSltValue	:= ADR(a_tyCurrRcp[1].diMinSltValue);
	p_ProdRcpCurrRcp1MaxSltValue	:= ADR(a_tyCurrRcp[1].diMaxSltValue);
	p_ProdRcpCurrRcp1Pitch			:= ADR(a_tyCurrRcp[1].diPitch);
	p_ProdRcpCurrRcp1McMod			:= ADR(a_tyCurrRcp[1].usiMcMod);
	p_ProdRcpCurrRcp1FlippedBrd		:= ADR(a_tyCurrRcp[1].usiFlippedBrd);
	p_ProdRcpCurrRcp1TopToBtm		:= ADR(a_tyCurrRcp[1].bTopToBtm);
	p_ProdRcpCurrRcp1LongBrd		:= ADR(a_tyCurrRcp[1].bLongBrd);
	p_ProdRcpCurrRcp1DisplayInfo	:= ADR(a_tyCurrRcp[1].sDisplayInfo);
	p_ProdRcpCurrRcp1LastModified	:= ADR(a_tyCurrRcp[1].dtLastModified);
	p_ProdRcpCurrRcp1Width2 		:= ADR(a_tyCurrRcp[1].diWidthInUM2);
	p_ProdRcpCurrRcp1WidthRear		:= ADR(a_tyCurrRcp[1].diWidthInUMRear);
	p_ProdRcpCurrRcp1PitchRear		:= ADR(a_tyCurrRcp[1].diPitchRear);
	p_ProdRcpCurrRcp1MinSltRear		:= ADR(a_tyCurrRcp[1].diMinSltValueRear);
	p_ProdRcpCurrRcp1MaxSltRear		:= ADR(a_tyCurrRcp[1].diMaxSltValueRear);
	p_ProdRcpCurrRcp1PshrOffset		:= ADR(a_tyCurrRcp[1].diPshrOffset);
	p_ProdRcpCurrRcp1MtrPshrExtSpd	:= ADR(a_tyCurrRcp[1].diMtrPshrExtSpd);
	p_ProdRcpCurrRcp1MtrPshrExtTorq	:= ADR(a_tyCurrRcp[1].diMtrPshrExtTorq);

	p_ProdRcpCurrRcp2				:= ADR(a_tyCurrRcp[2]);
	p_ProdRcpCurrRcp2Nm				:= ADR(a_tyCurrRcp[2].sRcpNm);
	p_ProdRcpCurrRcp2Width			:= ADR(a_tyCurrRcp[2].diWidthInUM);
	p_ProdRcpCurrRcp2MinSltValue	:= ADR(a_tyCurrRcp[2].diMinSltValue);
	p_ProdRcpCurrRcp2MaxSltValue	:= ADR(a_tyCurrRcp[2].diMaxSltValue);
	p_ProdRcpCurrRcp2Pitch			:= ADR(a_tyCurrRcp[2].diPitch);
	p_ProdRcpCurrRcp2McMod			:= ADR(a_tyCurrRcp[2].usiMcMod);
	p_ProdRcpCurrRcp2FlippedBrd		:= ADR(a_tyCurrRcp[2].usiFlippedBrd);
	p_ProdRcpCurrRcp2TopToBtm		:= ADR(a_tyCurrRcp[2].bTopToBtm);
	p_ProdRcpCurrRcp2LongBrd		:= ADR(a_tyCurrRcp[2].bLongBrd);
	p_ProdRcpCurrRcp2DisplayInfo	:= ADR(a_tyCurrRcp[2].sDisplayInfo);
	p_ProdRcpCurrRcp2LastModified	:= ADR(a_tyCurrRcp[2].dtLastModified);
	p_ProdRcpCurrRcp2Width2 		:= ADR(a_tyCurrRcp[2].diWidthInUM2);
	p_ProdRcpCurrRcp2WidthRear		:= ADR(a_tyCurrRcp[2].diWidthInUMRear);
	p_ProdRcpCurrRcp2PitchRear		:= ADR(a_tyCurrRcp[2].diPitchRear);
	p_ProdRcpCurrRcp2MinSltRear		:= ADR(a_tyCurrRcp[2].diMinSltValueRear);
	p_ProdRcpCurrRcp2MaxSltRear		:= ADR(a_tyCurrRcp[2].diMaxSltValueRear);
	p_ProdRcpCurrRcp2PshrOffset		:= ADR(a_tyCurrRcp[2].diPshrOffset);
	p_ProdRcpCurrRcp2MtrPshrExtSpd	:= ADR(a_tyCurrRcp[2].diMtrPshrExtSpd);
	p_ProdRcpCurrRcp2MtrPshrExtTorq	:= ADR(a_tyCurrRcp[2].diMtrPshrExtTorq);

	p_ProdRcpCurrRcp3				:= ADR(a_tyCurrRcp[3]);
	p_ProdRcpCurrRcp3Nm				:= ADR(a_tyCurrRcp[3].sRcpNm);
	p_ProdRcpCurrRcp3Width			:= ADR(a_tyCurrRcp[3].diWidthInUM);
	p_ProdRcpCurrRcp3MinSltValue	:= ADR(a_tyCurrRcp[3].diMinSltValue);
	p_ProdRcpCurrRcp3MaxSltValue	:= ADR(a_tyCurrRcp[3].diMaxSltValue);
	p_ProdRcpCurrRcp3Pitch			:= ADR(a_tyCurrRcp[3].diPitch);
	p_ProdRcpCurrRcp3McMod			:= ADR(a_tyCurrRcp[3].usiMcMod);
	p_ProdRcpCurrRcp3FlippedBrd		:= ADR(a_tyCurrRcp[3].usiFlippedBrd);
	p_ProdRcpCurrRcp3TopToBtm		:= ADR(a_tyCurrRcp[3].bTopToBtm);
	p_ProdRcpCurrRcp3LongBrd		:= ADR(a_tyCurrRcp[3].bLongBrd);
	p_ProdRcpCurrRcp3DisplayInfo	:= ADR(a_tyCurrRcp[3].sDisplayInfo);
	p_ProdRcpCurrRcp3LastModified	:= ADR(a_tyCurrRcp[3].dtLastModified);
	p_ProdRcpCurrRcp3Width2 		:= ADR(a_tyCurrRcp[3].diWidthInUM2);
	p_ProdRcpCurrRcp3WidthRear		:= ADR(a_tyCurrRcp[3].diWidthInUMRear);
	p_ProdRcpCurrRcp3PitchRear		:= ADR(a_tyCurrRcp[3].diPitchRear);
	p_ProdRcpCurrRcp3MinSltRear		:= ADR(a_tyCurrRcp[3].diMinSltValueRear);
	p_ProdRcpCurrRcp3MaxSltRear		:= ADR(a_tyCurrRcp[3].diMaxSltValueRear);
	p_ProdRcpCurrRcp3PshrOffset		:= ADR(a_tyCurrRcp[3].diPshrOffset);
	p_ProdRcpCurrRcp3MtrPshrExtSpd	:= ADR(a_tyCurrRcp[3].diMtrPshrExtSpd);
	p_ProdRcpCurrRcp3MtrPshrExtTorq	:= ADR(a_tyCurrRcp[3].diMtrPshrExtTorq);

	p_ProdRcpCurrRcp4				:= ADR(a_tyCurrRcp[4]);
	p_ProdRcpCurrRcp4Nm				:= ADR(a_tyCurrRcp[4].sRcpNm);
	p_ProdRcpCurrRcp4Width			:= ADR(a_tyCurrRcp[4].diWidthInUM);
	p_ProdRcpCurrRcp4MinSltValue	:= ADR(a_tyCurrRcp[4].diMinSltValue);
	p_ProdRcpCurrRcp4MaxSltValue	:= ADR(a_tyCurrRcp[4].diMaxSltValue);
	p_ProdRcpCurrRcp4Pitch			:= ADR(a_tyCurrRcp[4].diPitch);
	p_ProdRcpCurrRcp4McMod			:= ADR(a_tyCurrRcp[4].usiMcMod);
	p_ProdRcpCurrRcp4FlippedBrd		:= ADR(a_tyCurrRcp[4].usiFlippedBrd);
	p_ProdRcpCurrRcp4TopToBtm		:= ADR(a_tyCurrRcp[4].bTopToBtm);
	p_ProdRcpCurrRcp4LongBrd		:= ADR(a_tyCurrRcp[4].bLongBrd);
	p_ProdRcpCurrRcp4DisplayInfo	:= ADR(a_tyCurrRcp[4].sDisplayInfo);
	p_ProdRcpCurrRcp4LastModified	:= ADR(a_tyCurrRcp[4].dtLastModified);
	p_ProdRcpCurrRcp4Width2 		:= ADR(a_tyCurrRcp[4].diWidthInUM2);
	p_ProdRcpCurrRcp4WidthRear		:= ADR(a_tyCurrRcp[4].diWidthInUMRear);
	p_ProdRcpCurrRcp4PitchRear		:= ADR(a_tyCurrRcp[4].diPitchRear);
	p_ProdRcpCurrRcp4MinSltRear		:= ADR(a_tyCurrRcp[4].diMinSltValueRear);
	p_ProdRcpCurrRcp4MaxSltRear		:= ADR(a_tyCurrRcp[4].diMaxSltValueRear);
	p_ProdRcpCurrRcp4PshrOffset		:= ADR(a_tyCurrRcp[4].diPshrOffset);
	p_ProdRcpCurrRcp4MtrPshrExtSpd	:= ADR(a_tyCurrRcp[4].diMtrPshrExtSpd);
	p_ProdRcpCurrRcp4MtrPshrExtTorq	:= ADR(a_tyCurrRcp[4].diMtrPshrExtTorq);

	p_ProdRcpCurrRcp5				:= ADR(a_tyCurrRcp[5]);
	p_ProdRcpCurrRcp5Nm				:= ADR(a_tyCurrRcp[5].sRcpNm);
	p_ProdRcpCurrRcp5Width			:= ADR(a_tyCurrRcp[5].diWidthInUM);
	p_ProdRcpCurrRcp5MinSltValue	:= ADR(a_tyCurrRcp[5].diMinSltValue);
	p_ProdRcpCurrRcp5MaxSltValue	:= ADR(a_tyCurrRcp[5].diMaxSltValue);
	p_ProdRcpCurrRcp5Pitch			:= ADR(a_tyCurrRcp[5].diPitch);
	p_ProdRcpCurrRcp5McMod			:= ADR(a_tyCurrRcp[5].usiMcMod);
	p_ProdRcpCurrRcp5FlippedBrd		:= ADR(a_tyCurrRcp[5].usiFlippedBrd);
	p_ProdRcpCurrRcp5TopToBtm		:= ADR(a_tyCurrRcp[5].bTopToBtm);
	p_ProdRcpCurrRcp5LongBrd		:= ADR(a_tyCurrRcp[5].bLongBrd);
	p_ProdRcpCurrRcp5DisplayInfo	:= ADR(a_tyCurrRcp[5].sDisplayInfo);
	p_ProdRcpCurrRcp5LastModified	:= ADR(a_tyCurrRcp[5].dtLastModified);
	p_ProdRcpCurrRcp5Width2			:= ADR(a_tyCurrRcp[5].diWidthInUM2);
	p_ProdRcpCurrRcp5WidthRear		:= ADR(a_tyCurrRcp[5].diWidthInUMRear);
	p_ProdRcpCurrRcp5PitchRear		:= ADR(a_tyCurrRcp[5].diPitchRear);
	p_ProdRcpCurrRcp5MinSltRear		:= ADR(a_tyCurrRcp[5].diMinSltValueRear);
	p_ProdRcpCurrRcp5MaxSltRear		:= ADR(a_tyCurrRcp[5].diMaxSltValueRear);
	p_ProdRcpCurrRcp5PshrOffset		:= ADR(a_tyCurrRcp[5].diPshrOffset);
	p_ProdRcpCurrRcp5MtrPshrExtSpd	:= ADR(a_tyCurrRcp[5].diMtrPshrExtSpd);
	p_ProdRcpCurrRcp5MtrPshrExtTorq	:= ADR(a_tyCurrRcp[5].diMtrPshrExtTorq);
	(* Always Change If Project Change *)

END_PROGRAM
```

### Program Logical/MpProdRcp/MpProdRcp

#### Act_Alarm.st
```iecst
(** 2019-04-28 **)
ACTION Act_Alarm:

	//Error
	IF EDGEPOS(eStatus = Error) THEN

		tyAlmData.sProgNm		:= p_sProgNm;
		tyAlmData.udiCode		:= udiStatus;
		tyAlmData.eSeverity		:= AlmSeverityError;
		tyAlmData.udiRunTime	:= tyAlmData.udiRunTime + 1;
		tyAlmData.bAlm			:= TRUE;
		tyAlmData.udiModuleNum  := udiModuleNum;
		g_sMpProdRcpProgNm		:= p_sProgNm;
		//Get Error Message
		IF tyAlmData.udiCode < 10000 OR tyAlmData.udiCode > 10099 THEN
			tyAlmData.sAlmMsg	:= 'Unknown';
			tyAlmData.sRcyMsg	:= 'Unknown';
		ELSE
			tyAlmData.sAlmMsg	:= a_tyAlmText[tyAlmData.udiCode].sAlmText;
			tyAlmData.sRcyMsg	:= a_tyAlmText[tyAlmData.udiCode].sRcyText;
		END_IF

		sStatTxt	:= tyAlmData.sAlmMsg;

	ELSIF bRstErr AND (tyAlmData.udiCode <> 0) THEN

		tyAlmData.udiCode	:= 0;
		tyAlmData.eSeverity	:= AlmSeverityNA;
		tyAlmData.sAlmMsg	:= '';
		tyAlmData.sRcyMsg	:= '';
		tyAlmData.bAlm			:= FALSE;
		sStatTxt	:= a_sStatText[eStat];

	END_IF

END_ACTION
```

### MagRcp.typ - Change By Project
```iecst
(*2019-05-09*)
(**)
(*Action*)

TYPE
	eMagRcpAction :
		(
		MagRcpActIdle,
		MagRcpActCreateDir,
		MagRcpActAddEdit,
		MagRcpActDel,
		MagRcpActGetInfo,
		MagRcpActGetList,
		MagRcpActFilter,
		MagRcpActReadCurrRcp,
		MagRcpActLoadRcp,
		MagRcpActWriteCurrRcpParam,
		MagRcpActSaveList,
		MagRcpActSort
		);
END_TYPE

(**)
(*Data*)

TYPE
	tyMagRcpParam : 	STRUCT
		sRcpNm : STRING[30];
		diTtlSlt : DINT;
		diSltToSltInUM : DINT;
		diMag1Slt1PosInUM : DINT;
		diMag2Slt1PosInUM : DINT;
		diMag3Slt1PosInUM : DINT;
		diMag4Slt1PosInUM : DINT;
		diMag1TravPosInUM : DINT;
		diMag2TravPosInUM : DINT;
		diMag3TravPosInUM : DINT;
		diMag4TravPosInUM : DINT;
		usiMagModel : USINT; (*0=CAB706.2/1=CAB716.2/2=CAB717.2*)
		sDisplayInfo : STRING[30];
		diMagMaxBrdWidth : DINT;
		dtLastModified : DATE_AND_TIME;
		bSafetyBarDisabled : BOOL;
		bMagHeightChkEn : BOOL;
	END_STRUCT;
END_TYPE
```

### MagRcp.var - Change By Project
```iecst
(*2019-05-04*)
(**)
(*Constant*)
VAR CONSTANT
	c_udiMagRcpMax : UDINT := 10;
END_VAR
(**)
(*Action & State & Status*)
VAR
	p_MagRcpStat : UDINT;
	p_MagRcpStatus : UDINT;
	p_MagRcpStatTxt : UDINT;
END_VAR
(**)
(*Alarm*)
VAR
	p_MagRcpAlmData : UDINT;
END_VAR
(**)
(*Output*)
VAR
	p_MagRcpNmExist : UDINT;
	p_MagRcpNmNotExist : UDINT;
	p_MagRcpNmEmpty : UDINT;
	p_MagRcpListFull : UDINT;
	p_MagRcpCurrList : UDINT;
	p_MagRcpFilterList : UDINT;
	p_MagRcpSortedList : UDINT;
	p_MagRcpInfoOut : UDINT;
	p_MagRcpFileNotFound : UDINT;
	p_MagRcpCurrRcp : UDINT;
	p_MagRcpCurrRcpNm : UDINT;
	p_MagRcpCurrRcpTtlSlt : UDINT;
	p_MagRcpCurrRcpSltToSlt : UDINT;
	p_MagRcpCurrRcpMag1Slt1Pos : UDINT;
	p_MagRcpCurrRcpMag2Slt1Pos : UDINT;
	p_MagRcpCurrRcpMag3Slt1Pos : UDINT;
	p_MagRcpCurrRcpMag4Slt1Pos : UDINT;
	p_MagRcpCurrRcpMag1TravPos : UDINT;
	p_MagRcpCurrRcpMag2TravPos : UDINT;
	p_MagRcpCurrRcpMag3TravPos : UDINT;
	p_MagRcpCurrRcpMag4TravPos : UDINT;
	p_MagRcpCurrRcpDisplayInfo : UDINT;
	p_MagRcpCurrRcpMagMaxBrdWidth : UDINT;
	p_MagRcpCurrRcpLastModified : UDINT;
	p_MagRcpCurrRcpMagModel : UDINT;
	p_MagRcpCurrRcpSBarDisabled : UDINT;
	p_MagRcpCurrRcpMagHeightChkEn : UDINT;
END_VAR
(**)
```

### Program Logical/MagRcp/MagRcp (IEC) - 1.00.0 - NtRecipe v5.00.0 , NtFileIO v5.00.0

#### InputRef.var
```iecst
(*2020-07-24*)
(**)
(*General*)
VAR
	p_eAct : REFERENCE TO eMagRcpAction;
	p_udiMax : REFERENCE TO UDINT;
	p_udiRstErr : REFERENCE TO UDINT;
	p_bPrep : REFERENCE TO BOOL;
	p_bDis : REFERENCE TO BOOL;
END_VAR
(**)
(*Configuration*)
VAR
	p_dtCurrDT : REFERENCE TO DATE_AND_TIME;
	p_sSearch : REFERENCE TO STRING[30];
	p_tyInfoIn : REFERENCE TO tyMagRcpParam;
	p_tyCurrRcpWr : REFERENCE TO tyMagRcpParam;
	p_sListFileName : REFERENCE TO STRING[80];
	p_sSingleFileName : REFERENCE TO STRING[80];
	p_sProgNm : REFERENCE TO STRING[15];
	p_bNtSettingsLoadDone : REFERENCE TO BOOL;
END_VAR
```

#### Local.var
```iecst
(*2023-02-13*)
(**)
(*Local Action, State & Status*)
VAR
	eAct : eMagRcpAction := MagRcpActIdle;
	eStat : eMagRcpAction := MagRcpActIdle;
	eStatus : eFBStatus := Idle;
	udiStatus : UDINT := 0;
	sStatTxt : STRING[200] := '';
	a_sStatText : ARRAY[0..50] OF STRING[200] := ['Idling','Creating Directory','Adding and Editing Files','Deleting Files','Get Info','Get List','Filtering Files','Reading Current Recipe','Loading Current Recipe','Writing Current Recipe Parameter','Saving List',40('')];
END_VAR
(**)
(*Local Alarm*)
VAR
	tyAlmData : tyAlmDat;
	a_tyAlmText : ARRAY[10000..10099] OF tyAlmTxt := [(sAlmText:='Create User Directory Error',sRcyText:='Unable To Create User Directory. Please Contact Nutek For A Possible Solution'),(sAlmText:='Create Magazine Recipe Directory Error',sRcyText:='Unable To Create Magazine Recipe Directory. Please Contact Nutek For A Possible Solution'),(sAlmText:='File Open Error While Adding & Editing',sRcyText:='An Error Was Encountered While Trying To Open File. Please Contact Nutek For A Possible Solution.'),(sAlmText:='File Create Error While Adding & Editing',sRcyText:='An Error Was Encountered While Trying To Create File. Please Contact Nutek For A Possible Solution.'),(sAlmText:='File Write Error While Adding & Editing',sRcyText:='An Error Was Encountered While Trying To Write File. Please Contact Nutek For A Possible Solution.'),(sAlmText:='File Close Error While Adding & Editing',sRcyText:='An Error Was Encountered While Trying To Close File. Please Contact Nutek For A Possible Solution.'),(sAlmText:='File Open Error While Deleting',sRcyText:='An Error Was Encountered While Trying To Open File. Please Contact Nutek For A Possible Solution.'),(sAlmText:='File Create Error While Deleting',sRcyText:='An Error Was Encountered While Trying To Create File. Please Contact Nutek For A Possible Solution.'),(sAlmText:='File Write Error While Deleting',sRcyText:='An Error Was Encountered While Trying To Write File. Please Contact Nutek For A Possible Solution.'),(sAlmText:='File Close Error While Deleting',sRcyText:='An Error Was Encountered While Trying To Close File. Please Contact Nutek For A Possible Solution.'),(sAlmText:='File Open Error While Getting List',sRcyText:='An Error Was Encountered While Trying To Open File. Please Contact Nutek For A Possible Solution.'),(sAlmText:='File Read Error While Getting List',sRcyText:='An Error Was Encountered While Trying To Read File. Please Contact Nutek For A Possible Solution.'),(sAlmText:='File Close Error While Getting List',sRcyText:='An Error Was Encountered While Trying To Close File. Please Contact Nutek For A Possible Solution.'),(sAlmText:='Directory Does Not Exist While Adding & Editing',sRcyText:='The Directory Does Not Exist.Please Contact Nutek For A Possible Solution.'),(sAlmText:='Directory Does Not Exist While Deleting',sRcyText:='The Directory Does Not Exist.Please Contact Nutek For A Possible Solution.'),(sAlmText:='File Open Error While Loading Current Recipe',sRcyText:='An Error Was Encountered While Trying To Open File. Please Contact Nutek For A Possible Solution.'),(sAlmText:='File Create Error While Loading Current Recipe',sRcyText:='An Error Was Encountered While Trying To Create File. Please Contact Nutek For A Possible Solution.'),(sAlmText:='File Write Error While Loading Current Recipe',sRcyText:='An Error Was Encountered While Trying To Write File. Please Contact Nutek For A Possible Solution.'),(sAlmText:='File Close Error While Loading Current Recipe',sRcyText:='An Error Was Encountered While Trying To Close File. Please Contact Nutek For A Possible Solution.'),(sAlmText:='Directory Does Not Exist While Loading Current Recipe',sRcyText:='The Directory Does Not Exist.Please Contact Nutek For A Possible Solution.'),(sAlmText:='File Open Error While Reading Current Recipe',sRcyText:='An Error Was Encountered While Trying To Open File. Please Contact Nutek For A Possible Solution.'),(sAlmText:='File Read Error While Reading Current Recipe',sRcyText:='An Error Was Encountered While Trying To Read File. Please Contact Nutek For A Possible Solution.'),(sAlmText:='File Close Error While Reading Current Recipe',sRcyText:='An Error Was Encountered While Trying To Close File. Please Contact Nutek For A Possible Solution.'),(sAlmText:='File Open Error While Writing Current Recipe Parameter',sRcyText:='An Error Was Encountered While Trying To Open File. Please Contact Nutek For A Possible Solution.'),(sAlmText:='File Create Error While Writing Current Recipe Parameter',sRcyText:='An Error Was Encountered While Trying To Create File. Please Contact Nutek For A Possible Solution.'),(sAlmText:='File Write Error While Writing Current Recipe Parameter',sRcyText:='An Error Was Encountered While Trying To Write File. Please Contact Nutek For A Possible Solution.'),(sAlmText:='File Close Error While Writing Current Recipe Parameter',sRcyText:='An Error Was Encountered While Trying To Close File. Please Contact Nutek For A Possible Solution.'),(sAlmText:='Directory Does Not Exist While Writing Current Recipe Parameter',sRcyText:='The Directory Does Not Exist.Please Contact Nutek For A Possible Solution.'),(sAlmText:='File Open Error While Saving List',sRcyText:='An Error Was Encountered While Trying To Open File. Please Contact Nutek For A Possible Solution.'),(sAlmText:='File Create Error While Saving List',sRcyText:='An Error Was Encountered While Trying To Create File. Please Contact Nutek For A Possible Solution.'),(sAlmText:='File Write Error While Saving List',sRcyText:='An Error Was Encountered While Trying To Write File. Please Contact Nutek For A Possible Solution.'),(sAlmText:='File Close Error While Saving List',sRcyText:='An Error Was Encountered While Trying To Close File. Please Contact Nutek For A Possible Solution.'),(sAlmText:='Directory Does Not Exist While Saving List',sRcyText:='The Directory Does Not Exist.Please Contact Nutek For A Possible Solution.'),67(0)];
END_VAR
(**)
(*Local Output*)
VAR
	bNmExist : BOOL;
	bNmNotExist : BOOL;
	bNmEmpty : BOOL;
	bListFull : BOOL;
	a_tyCurrList : ARRAY[1..c_udiMagRcpMax] OF tyMagRcpParam;
	a_tyFilterList : ARRAY[1..c_udiMagRcpMax] OF tyMagRcpParam;
	a_tySortList : ARRAY[1..c_udiMagRcpMax] OF tyMagRcpParam;
	tyTempList : tyMagRcpParam;
	tyInfoOut : tyMagRcpParam;
	bFileNotFound : BOOL;
	tyCurrRcp : tyMagRcpParam;
END_VAR
(**)
(*Local Input*)
VAR
	udiRstErr : UDINT := 0;
	bPrep : BOOL := TRUE;
	bDis : BOOL := FALSE;
	dtCurrDT : DATE_AND_TIME;
	sSearch : STRING[254] := '';
	tyInfoIn : tyMagRcpParam;
	tyCurrRcpWr : tyMagRcpParam;
	sListFileName : STRING[80] := 'MagazineRecipeList.dat';
	sSingleFileName : STRING[80] := 'MagazineRecipe.dat';
	sProgNm : STRING[15] := 'MagRcp';
	bNtSettingsLoadDone : BOOL := TRUE;
	udiSortCurrenTotalCntr : UDINT;
	iSortCurrentInnerCntr : INT;
	iSortCurrentOuterCntr : INT;
	iTotalRcp : INT;
	i : {REDUND_UNREPLICABLE} INT;
	udi : UDINT;
	sDebug : STRING[300];
	tyTempRecipe : tyMagRcpParam;
END_VAR
(**)
(*Local*)
VAR
	bRstErr : BOOL;
	udiRstErrOld : UDINT;
	bInitDone : BOOL;
	bInitialDone : BOOL;
	usiStep : USINT;
	udiAddStatus : UDINT;
	a_tyListTemp : ARRAY[1..c_udiMagRcpMax] OF tyMagRcpParam;
	fbDirCreate1 : fbDirCreate;
	fbDirCreate2 : fbDirCreate;
	fbFileReadList : fbFileFullRead;
	fbFileWriteList : fbFileFullWrite;
	fbFileReadSingle : fbFileFullRead;
	fbFileWriteSingle : fbFileFullWrite;
	fbFileLoadSingle : fbFileFullWrite;
	iFilterCtr : INT;
	udiModuleNum : UDINT := 4901;
END_VAR
```

#### Act_InitGlobal.st
```iecst
(** 2019-03-25 **)
ACTION Act_InitGlobal:

	(* Always Change If Project Change *)

	//Pass Data To Link
	p_bLinkStartupRun ACCESS p_StartupRun;

	//Pass Data To Internal Use
	p_udiRstErr ACCESS p_RstErrReset;
	p_dtCurrDT ACCESS p_TimeCurrDT;
	p_sSearch ACCESS p_UIMagRcpSearch;
	p_tyInfoIn ACCESS p_UIMagRcpInfoIn;
	p_sListFileName ACCESS p_NtParamMagRcpListFileNm;
	p_sSingleFileName ACCESS p_NtParamMagRcpSingleFileNm;
	p_sProgNm ACCESS p_NtParamMagRcpProgNm;
	p_bNtSettingsLoadDone ACCESS p_StartupNtSettingsLoadDone;

	(* Always Change If Project Change *)

END_ACTION
```

#### Act_LinkAction.st
```iecst
(** 2019-03-29 **)
ACTION Act_LinkAction:

	IF p_bLinkStartupRun = TRUE THEN
		p_eAct ACCESS p_StartupMagRcpAct;
	ELSE
		p_eAct ACCESS p_UIMagRcpAct;
	END_IF

END_ACTION
```

#### Act_Main.st
```iecst
(** 2023-02-13 **)
ACTION Act_Main:

	//Main
	CASE eStat OF

		MagRcpActIdle:
			IF eStatus <> Idle THEN	//Reset Data
				//Private
				fbDirCreate1(bEn := FALSE);
				fbDirCreate2(bEn := FALSE);
				fbFileReadList(bEn := FALSE);
				fbFileWriteList(bEn := FALSE);
				fbFileReadSingle(bEn := FALSE);
				fbFileWriteSingle(bEn := FALSE);
				usiStep			:= 0;
				udiAddStatus	:= 0;

				bNmExist		:= FALSE;
				bNmNotExist		:= FALSE;
				bNmEmpty		:= FALSE;
				bListFull		:= FALSE;
				bFileNotFound	:= FALSE;
				iTotalRcp		:= 0;

				memset(ADR(tyTempRecipe), 0 , SIZEOF(tyTempRecipe));

				sStatTxt	:= a_sStatText[eStat];

			END_IF

			eStatus	:= Idle;

		MagRcpActCreateDir:
			IF eStatus = Idle OR eStatus = Busy THEN

				eStatus	:= Busy;

				sStatTxt	:= a_sStatText[eStat];

				CASE usiStep OF
					0:
						fbDirCreate1(bEn := TRUE);
						IF fbDirCreate1.udiStatus = 0 THEN
							usiStep	:= 1;
						ELSIF fbDirCreate1.udiStatus < 65534 THEN
							eStatus		:= Error;

							IF fbDirCreate1.udiStatus = 1908 THEN
								udiStatus	:= 10000;	//Create User Directory Error
							ELSE
								udiStatus	:= fbDirCreate1.udiStatus;
							END_IF
						END_IF

					1:
						fbDirCreate2(bEn := TRUE);
						IF fbDirCreate2.udiStatus = 0 THEN
							eStatus	:= Done;
						ELSIF fbDirCreate2.udiStatus < 65534 THEN
							eStatus		:= Error;

							IF fbDirCreate2.udiStatus = 1908 THEN
								udiStatus	:= 10001;	//Create Magazine Recipe Directory Error
							ELSE
								udiStatus	:= fbDirCreate2.udiStatus;
							END_IF
						END_IF

				END_CASE

			END_IF

		MagRcpActAddEdit:
			IF eStatus = Idle OR eStatus = Busy THEN

				eStatus	:= Busy;

				sStatTxt	:= a_sStatText[eStat];

				CASE usiStep OF
					0:	//Edit Recipe
						udiAddStatus	:= fRecipeAddEdit(ADR(p_tyInfoIn) , ADR(a_tyListTemp) , SIZEOF(a_tyListTemp[1]) , ADR(a_tyListTemp[1].sRcpNm) , SIZEOF(a_tyListTemp[1].sRcpNm) , p_udiMax);

						IF udiAddStatus = 1600 THEN	//Recipe Name Empty
							bNmEmpty	:= TRUE;
							eStatus		:= Done;

						ELSIF udiAddStatus = 1601 THEN	//Recipe Full
							bListFull	:= TRUE;
							eStatus		:= Done;

						ELSIF udiAddStatus = 0 THEN	//OK
							usiStep	:= 1;

						END_IF

					1:	//Write Into File
						fbFileWriteList(bEn := TRUE);

						IF fbFileWriteList.udiStatus = 0 THEN
							a_tyCurrList	:= a_tyListTemp;
							eStatus			:= Done;

						ELSIF fbFileWriteList.udiStatus < 65534 THEN
							a_tyListTemp	:= a_tyCurrList;
							eStatus			:= Error;

							IF fbFileWriteList.udiStatus = 1900 THEN
								udiStatus	:= 10002;	//File Open Error While Adding & Editing
							ELSIF fbFileWriteList.udiStatus = 1901 THEN
								udiStatus	:= 10003;	//File Create Error While Adding & Editing
							ELSIF fbFileWriteList.udiStatus = 1903 THEN
								udiStatus	:= 10004;	//File Write Error While Adding & Editing
							ELSIF fbFileWriteList.udiStatus = 1904 THEN
								udiStatus	:= 10005;	//File Close Error While Adding & Editing
							ELSIF fbFileWriteList.udiStatus = 1914 THEN
								udiStatus	:= 10013;	//Directory Does Not Exist While Adding & Editing
							ELSE
								udiStatus	:= fbFileWriteList.udiStatus;
							END_IF
						END_IF

				END_CASE

			END_IF

		MagRcpActDel:
			IF eStatus = Idle OR eStatus = Busy THEN

				eStatus	:= Busy;

				sStatTxt	:= a_sStatText[eStat];

				CASE usiStep OF
					0:	//Delete Recipe
						udiAddStatus	:= fRecipeDelete(ADR(p_tyInfoIn) , ADR(a_tyListTemp) , SIZEOF(a_tyListTemp[1]) , ADR(a_tyListTemp[1].sRcpNm) , SIZEOF(a_tyListTemp[1].sRcpNm) , p_udiMax);

						IF udiAddStatus = 1600 THEN	//Recipe Name Empty
							bNmEmpty	:= TRUE;
							eStatus		:= Done;

						ELSIF udiAddStatus = 1603 THEN	//Recipe Not Exist
							bNmNotExist	:= TRUE;
							eStatus		:= Done;

						ELSIF udiAddStatus = 0 THEN	//OK
							usiStep	:= 1;

						END_IF

					1:	//Write Into File
						fbFileWriteList(bEn := TRUE);

						IF fbFileWriteList.udiStatus = 0 THEN
							a_tyCurrList	:= a_tyListTemp;
							eStatus			:= Done;

						ELSIF fbFileWriteList.udiStatus < 65534 THEN
							a_tyListTemp	:= a_tyCurrList;
							eStatus			:= Error;

							IF fbFileWriteList.udiStatus = 1900 THEN
								udiStatus	:= 10006;	//File Open Error While Deleting
							ELSIF fbFileWriteList.udiStatus = 1901 THEN
								udiStatus	:= 10007;	//File Create Error While Deleting
							ELSIF fbFileWriteList.udiStatus = 1903 THEN
								udiStatus	:= 10008;	//File Write Error While Deleting
							ELSIF fbFileWriteList.udiStatus = 1904 THEN
								udiStatus	:= 10009;	//File Close Error While Deleting
							ELSIF fbFileWriteList.udiStatus = 1914 THEN
								udiStatus	:= 10014;	//Directory Does Not Exist While Deleting
							ELSE
								udiStatus	:= fbFileWriteList.udiStatus;
							END_IF
						END_IF

				END_CASE

			END_IF

		MagRcpActGetInfo:
			IF eStatus = Idle OR eStatus = Busy THEN

				sStatTxt	:= a_sStatText[eStat];

				IF p_tyInfoIn.sRcpNm = '' THEN
					bNmEmpty	:= TRUE;
					bNmNotExist	:= TRUE;
				ELSE
					bNmNotExist	:= (fRecipeGetInfo(p_tyInfoIn.sRcpNm , ADR(tyInfoOut) , ADR(a_tyCurrList) , SIZEOF(a_tyCurrList[1]) , ADR(a_tyCurrList[1].sRcpNm) , SIZEOF(a_tyCurrList[1].sRcpNm) , p_udiMax)) = 0;
				END_IF

				eStatus	:= Done;

			END_IF

		MagRcpActGetList:
			IF eStatus = Idle OR eStatus = Busy THEN

				eStatus	:= Busy;

				sStatTxt	:= a_sStatText[eStat];

				fbFileReadList(bEn := TRUE);
				IF fbFileReadList.udiStatus = 0 THEN
					a_tyListTemp	:= a_tyCurrList;
					eStatus			:= Done;

				ELSIF fbFileReadList.udiStatus < 65534 THEN
					eStatus		:= Error;

					IF fbFileReadList.udiStatus = 1900 THEN
						udiStatus	:= 10010;	//File Open Error While Getting List
					ELSIF fbFileReadList.udiStatus = 1902 THEN
						udiStatus	:= 10011;	//File Read Error While Getting List
					ELSIF fbFileReadList.udiStatus = 1904 THEN
						udiStatus	:= 10012;	//File Close Error While Getting List
					ELSIF fbFileReadList.udiStatus = 1915 THEN
						bFileNotFound	:= TRUE;
						eStatus			:= Done;
					ELSE
						udiStatus	:= fbFileReadList.udiStatus;
					END_IF
				END_IF

			END_IF

		MagRcpActFilter:
			IF eStatus = Idle OR eStatus = Busy THEN

				eStatus 	:= Busy;
				sStatTxt	:= a_sStatText[eStat];

				CASE usiStep OF
					0:
						fRecipeFilter(p_sSearch , ADR(a_tyFilterList) , ADR(a_tyCurrList) , SIZEOF(a_tyCurrList[1]) , ADR(a_tyCurrList[1].sRcpNm) ,
						SIZEOF(a_tyCurrList[1].sRcpNm) , p_udiMax, 0, 499, iFilterCtr);
						usiStep := 1;
					1:
						fRecipeFilter(p_sSearch , ADR(a_tyFilterList) , ADR(a_tyCurrList) , SIZEOF(a_tyCurrList[1]) , ADR(a_tyCurrList[1].sRcpNm) ,
						SIZEOF(a_tyCurrList[1].sRcpNm) , p_udiMax, 500, 999, iFilterCtr);
						usiStep := 2;
					2:
						fRecipeFilter(p_sSearch , ADR(a_tyFilterList) , ADR(a_tyCurrList) , SIZEOF(a_tyCurrList[1]) , ADR(a_tyCurrList[1].sRcpNm) ,
						SIZEOF(a_tyCurrList[1].sRcpNm) , p_udiMax, 1000, 1499, iFilterCtr);
						usiStep := 3;
					3:
						fRecipeFilter(p_sSearch , ADR(a_tyFilterList) , ADR(a_tyCurrList) , SIZEOF(a_tyCurrList[1]) , ADR(a_tyCurrList[1].sRcpNm) ,
						SIZEOF(a_tyCurrList[1].sRcpNm) , p_udiMax, 1500, 1999, iFilterCtr);
						eStatus := Done;

				END_CASE

			END_IF

		MagRcpActLoadRcp:
			IF eStatus = Idle OR eStatus = Busy THEN

				sStatTxt	:= a_sStatText[eStat];

				CASE usiStep OF
					0:	//Get Recipe
						IF p_tyInfoIn.sRcpNm = '' THEN
							bNmEmpty	:= TRUE;
							bNmNotExist	:= TRUE;

							eStatus	:= Done;
						ELSE
							bNmNotExist	:= (fRecipeGetInfo(p_tyInfoIn.sRcpNm , ADR(tyCurrRcp) , ADR(a_tyCurrList) , SIZEOF(a_tyCurrList[1]) , ADR(a_tyCurrList[1].sRcpNm) , SIZEOF(a_tyCurrList[1].sRcpNm) , p_udiMax)) = 0;
							IF bNmNotExist = TRUE THEN
								eStatus	:= Done;
							ELSE
								usiStep	:= 1;
							END_IF
						END_IF

					1:	//Write Into File
						fbFileLoadSingle(bEn := TRUE);

						IF fbFileLoadSingle.udiStatus = 0 THEN
							eStatus			:= Done;
						ELSIF fbFileLoadSingle.udiStatus < 65534 THEN
							eStatus			:= Error;

							IF fbFileLoadSingle.udiStatus = 1900 THEN
								udiStatus	:= 10015;	//File Open Error While Loading Current Recipe
							ELSIF fbFileLoadSingle.udiStatus = 1901 THEN
								udiStatus	:= 10016;	//File Create Error While Loading Current Recipe
							ELSIF fbFileLoadSingle.udiStatus = 1903 THEN
								udiStatus	:= 10017;	//File Write Error While Loading Current Recipe
							ELSIF fbFileLoadSingle.udiStatus = 1904 THEN
								udiStatus	:= 10018;	//File Close Error While Loading Current Recipe
							ELSIF fbFileLoadSingle.udiStatus = 1914 THEN
								udiStatus	:= 10019;	//Directory Does Not Exist While Loading Current Recipe
							ELSE
								udiStatus	:= fbFileLoadSingle.udiStatus;
							END_IF
						END_IF

				END_CASE

			END_IF

		MagRcpActReadCurrRcp:
			IF eStatus = Idle OR eStatus = Busy THEN

				eStatus	:= Busy;

				sStatTxt	:= a_sStatText[eStat];

				fbFileReadSingle(bEn := TRUE);
				IF fbFileReadSingle.udiStatus = 0 THEN
					eStatus	:= Done;

				ELSIF fbFileReadSingle.udiStatus < 65534 THEN
					eStatus		:= Error;

					IF fbFileReadSingle.udiStatus = 1900 THEN
						udiStatus	:= 10020;	//File Open Error While Reading Current Recipe
					ELSIF fbFileReadSingle.udiStatus = 1902 THEN
						udiStatus	:= 10021;	//File Read Error While Reading Current Recipe
					ELSIF fbFileReadSingle.udiStatus = 1904 THEN
						udiStatus	:= 10022;	//File Close Error While Reading Current Recipe
					ELSIF fbFileReadSingle.udiStatus = 1915 THEN
						bFileNotFound	:= TRUE;
						eStatus			:= Done;
					ELSE
						udiStatus	:= fbFileReadSingle.udiStatus;
					END_IF
				END_IF

			END_IF

		MagRcpActWriteCurrRcpParam:
			IF eStatus = Idle OR eStatus = Busy THEN

				sStatTxt	:= a_sStatText[eStat];

				fbFileWriteSingle(bEn := TRUE);

				IF fbFileWriteSingle.udiStatus = 0 THEN
					tyCurrRcp		:= p_tyCurrRcpWr;
					eStatus			:= Done;
				ELSIF fbFileWriteSingle.udiStatus < 65534 THEN
					eStatus			:= Error;

					IF fbFileWriteSingle.udiStatus = 1900 THEN
						udiStatus	:= 10023;	//File Open Error While Writing Current Recipe Parameter
					ELSIF fbFileWriteSingle.udiStatus = 1901 THEN
						udiStatus	:= 10024;	//File Create Error While Writing Current Recipe Parameter
					ELSIF fbFileWriteSingle.udiStatus = 1903 THEN
						udiStatus	:= 10025;	//File Write Error While Writing Current Recipe Parameter
					ELSIF fbFileWriteSingle.udiStatus = 1904 THEN
						udiStatus	:= 10026;	//File Close Error While Writing Current Recipe Parameter
					ELSIF fbFileWriteSingle.udiStatus = 1914 THEN
						udiStatus	:= 10027;	//Directory Does Not Exist While Writing Current Recipe Parameter
					ELSE
						udiStatus	:= fbFileWriteSingle.udiStatus;
					END_IF
				END_IF

			END_IF

		MagRcpActSaveList:
			IF eStatus = Idle OR eStatus = Busy THEN

				eStatus	:= Busy;

				sStatTxt	:= a_sStatText[eStat];

				CASE usiStep OF

					0:
						a_tyListTemp	:= a_tyCurrList;

						fbFileWriteList(bEn := TRUE);

						IF fbFileWriteList.udiStatus = 0 THEN
							eStatus			:= Done;

						ELSIF fbFileWriteList.udiStatus < 65534 THEN
							eStatus			:= Error;

							IF fbFileWriteList.udiStatus = 1900 THEN
								udiStatus	:= 10028;	//File Open Error While Saving List
							ELSIF fbFileWriteList.udiStatus = 1901 THEN
								udiStatus	:= 10029;	//File Create Error While Saving List
							ELSIF fbFileWriteList.udiStatus = 1903 THEN
								udiStatus	:= 10030;	//File Write Error While Saving List
							ELSIF fbFileWriteList.udiStatus = 1904 THEN
								udiStatus	:= 10031;	//File Close Error While Saving List
							ELSIF fbFileWriteList.udiStatus = 1914 THEN
								udiStatus	:= 10032;	//Directory Does Not Exist While Saving List
							ELSE
								udiStatus	:= fbFileWriteList.udiStatus;
							END_IF
						END_IF

				END_CASE

			END_IF

		MagRcpActSort:
			IF eStatus = Idle OR eStatus = Busy THEN

				eStatus 	:= Busy;

				sStatTxt	:= a_sStatText[eStat];

				CASE usiStep OF

					0:

						FOR udi := 1 TO c_udiMagRcpMax DO
							IF p_sSearch <> '' THEN
								IF a_tyFilterList[udi].sRcpNm = '' THEN
									usiStep := 1;
									EXIT;
								ELSIF udi = c_udiMagRcpMax THEN
									iTotalRcp := UDINT_TO_INT(c_udiMagRcpMax);
									usiStep := 1;
									EXIT;
								ELSE
									iTotalRcp := iTotalRcp +1;
								END_IF
							ELSE
								IF a_tyCurrList[udi].sRcpNm = '' THEN
									usiStep := 1;
									EXIT;
								ELSIF udi = c_udiMagRcpMax THEN
									iTotalRcp := UDINT_TO_INT(c_udiMagRcpMax);
									usiStep := 1;
									EXIT;
								ELSE
									iTotalRcp := iTotalRcp +1;
								END_IF
							END_IF
						END_FOR

					1:
						IF p_sSearch <> '' THEN
							memcpy(ADR(a_tySortList),ADR(a_tyFilterList), SIZEOF(a_tyFilterList));
						ELSE
							memcpy(ADR(a_tySortList),ADR(a_tyCurrList), SIZEOF(a_tyCurrList));
						END_IF

						iSortCurrentOuterCntr	:= 0;
						iSortCurrentInnerCntr	:= 1 ;

						udiSortCurrenTotalCntr	:= 0;

						usiStep := 2;

					2:

						IF iSortCurrentOuterCntr < iTotalRcp THEN

							FOR iSortCurrentInnerCntr:= iSortCurrentOuterCntr+1 TO iTotalRcp-1 DO

								IF fRecipeNmCompare(ADR(a_tySortList[iSortCurrentOuterCntr+1].sRcpNm),ADR(a_tySortList[iSortCurrentInnerCntr+1].sRcpNm),SIZEOF(a_tySortList[1].sRcpNm),ADR(sDebug)) THEN

									memcpy(ADR(tyTempRecipe), ADR(a_tySortList[iSortCurrentOuterCntr+1]), SIZEOF(a_tySortList[1]));
									memcpy(ADR(a_tySortList[iSortCurrentOuterCntr+1]), ADR(a_tySortList[iSortCurrentInnerCntr+1]), SIZEOF(a_tySortList[1]));
									memcpy(ADR(a_tySortList[iSortCurrentInnerCntr+1]), ADR(tyTempRecipe), SIZEOF(a_tySortList[1]));

								END_IF

								udiSortCurrenTotalCntr	:= udiSortCurrenTotalCntr + 1;

							END_FOR

							iSortCurrentOuterCntr	:= iSortCurrentOuterCntr + 1;

						ELSE
							usiStep := 3;
						END_IF

					3:
						eStatus	:= Done;

				END_CASE

			END_IF

	END_CASE

END_ACTION
```

#### Init.st
```iecst
(** 2019-05-04 **)
PROGRAM _INIT

	(* Always Change If Project Change *)

	//Pass Address To Global Address For External Use
	//Action, State & Status
	p_MagRcpStat	:= ADR(eStat);
	p_MagRcpStatus	:= ADR(eStatus);
	p_MagRcpStatTxt	:= ADR(sStatTxt);

	//Alarm
	p_MagRcpAlmData	:= ADR(tyAlmData);

	//Output
	p_MagRcpNmExist			:= ADR(bNmExist);
	p_MagRcpNmNotExist		:= ADR(bNmNotExist);
	p_MagRcpNmEmpty			:= ADR(bNmEmpty);
	p_MagRcpListFull		:= ADR(bListFull);
	p_MagRcpCurrList		:= ADR(a_tyCurrList);
	p_MagRcpFilterList		:= ADR(a_tyFilterList);
	p_MagRcpSortedList		:= ADR(a_tySortList);
	p_MagRcpInfoOut			:= ADR(tyInfoOut);
	p_MagRcpFileNotFound	:= ADR(bFileNotFound);

	p_MagRcpCurrRcp				:= ADR(tyCurrRcp);
	p_MagRcpCurrRcpNm			:= ADR(tyCurrRcp.sRcpNm);
	p_MagRcpCurrRcpTtlSlt		:= ADR(tyCurrRcp.diTtlSlt);
	p_MagRcpCurrRcpSltToSlt		:= ADR(tyCurrRcp.diSltToSltInUM);
	p_MagRcpCurrRcpMag1Slt1Pos	:= ADR(tyCurrRcp.diMag1Slt1PosInUM);
	p_MagRcpCurrRcpMag2Slt1Pos	:= ADR(tyCurrRcp.diMag2Slt1PosInUM);
	p_MagRcpCurrRcpMag3Slt1Pos	:= ADR(tyCurrRcp.diMag3Slt1PosInUM);
	p_MagRcpCurrRcpMag4Slt1Pos	:= ADR(tyCurrRcp.diMag4Slt1PosInUM);
	p_MagRcpCurrRcpMag1TravPos	:= ADR(tyCurrRcp.diMag1TravPosInUM);
	p_MagRcpCurrRcpMag2TravPos	:= ADR(tyCurrRcp.diMag2TravPosInUM);
	p_MagRcpCurrRcpMag3TravPos	:= ADR(tyCurrRcp.diMag3TravPosInUM);
	p_MagRcpCurrRcpMag4TravPos	:= ADR(tyCurrRcp.diMag4TravPosInUM);
	p_MagRcpCurrRcpDisplayInfo	:= ADR(tyCurrRcp.sDisplayInfo);
	p_MagRcpCurrRcpLastModified	:= ADR(tyCurrRcp.dtLastModified);
	p_MagRcpCurrRcpMagMaxBrdWidth	:= ADR(tyCurrRcp.diMagMaxBrdWidth);
	p_MagRcpCurrRcpMagModel		:= ADR(tyCurrRcp.usiMagModel);
	p_MagRcpCurrRcpSBarDisabled	:= ADR(tyCurrRcp.bSafetyBarDisabled);
	p_MagRcpCurrRcpMagHeightChkEn	:= ADR(tyCurrRcp.bMagHeightChkEn);
	(* Always Change If Project Change *)

END_PROGRAM
```

### MagRcp1.var - Change By Project
```iecst
(*2019-05-04*)
(**)
(*Constant*)
VAR CONSTANT
	c_udiMagRcpMax1 : UDINT := 10;
END_VAR
(**)
(*Action & State & Status*)
VAR
	p_MagRcpStat1 : UDINT;
	p_MagRcpStatus1 : UDINT;
	p_MagRcpStatTxt1 : UDINT;
END_VAR
(**)
(*Alarm*)
VAR
	p_MagRcpAlmData1 : UDINT;
END_VAR
(**)
(*Output*)
VAR
	p_MagRcpNmExist1 : UDINT;
	p_MagRcpNmNotExist1 : UDINT;
	p_MagRcpNmEmpty1 : UDINT;
	p_MagRcpListFull1 : UDINT;
	p_MagRcpCurrList1 : UDINT;
	p_MagRcpFilterList1 : UDINT;
	p_MagRcpSortedList1 : UDINT;
	p_MagRcpInfoOut1 : UDINT;
	p_MagRcpFileNotFound1 : UDINT;
	p_MagRcpCurrRcp1 : UDINT;
	p_MagRcpCurrRcpNm1 : UDINT;
	p_MagRcpCurrRcpTtlSlt1 : UDINT;
	p_MagRcpCurrRcpSltToSlt1 : UDINT;
	p_MagRcpCurrRcpMag1Slt1Pos1 : UDINT;
	p_MagRcpCurrRcpMag2Slt1Pos1 : UDINT;
	p_MagRcpCurrRcpMag3Slt1Pos1 : UDINT;
	p_MagRcpCurrRcpMag4Slt1Pos1 : UDINT;
	p_MagRcpCurrRcpMag1TravPos1 : UDINT;
	p_MagRcpCurrRcpMag2TravPos1 : UDINT;
	p_MagRcpCurrRcpMag3TravPos1 : UDINT;
	p_MagRcpCurrRcpMag4TravPos1 : UDINT;
	p_MagRcpCurrRcpDisplayInfo1 : UDINT;
	p_MagRcpCurrRcpMagMaxBrdWidth1 : UDINT;
	p_MagRcpCurrRcpLastModified1 : UDINT;
	p_MagRcpCurrRcpMagModel1 : UDINT;
	p_MagRcpCurrRcpSBarDisabled1 : UDINT;
	p_MagRcpCurrRcpMagHeightChkEn1 : UDINT;
END_VAR
(**)
```

### Program Logical/MagRcp/MagRcp1 (IEC) - 1.00.0 - NtRecipe v5.00.0 , NtFileIO v5.00.0

#### InputRef.var
```iecst
(*2020-07-24*)
(**)
(*General*)
VAR
	p_eAct : REFERENCE TO eMagRcpAction;
	p_udiMax : REFERENCE TO UDINT;
	p_udiRstErr : REFERENCE TO UDINT;
	p_bPrep : REFERENCE TO BOOL;
	p_bDis : REFERENCE TO BOOL;
END_VAR
(**)
(*Configuration*)
VAR
	p_dtCurrDT : REFERENCE TO DATE_AND_TIME;
	p_sSearch : REFERENCE TO STRING[254];
	p_tyInfoIn : REFERENCE TO tyMagRcpParam;
	p_tyCurrRcpWr : REFERENCE TO tyMagRcpParam;
	p_sListFileName : REFERENCE TO STRING[80];
	p_sSingleFileName : REFERENCE TO STRING[80];
	p_sProgNm : REFERENCE TO STRING[15];
	p_bNtSettingsLoadDone : REFERENCE TO BOOL;
END_VAR
```
